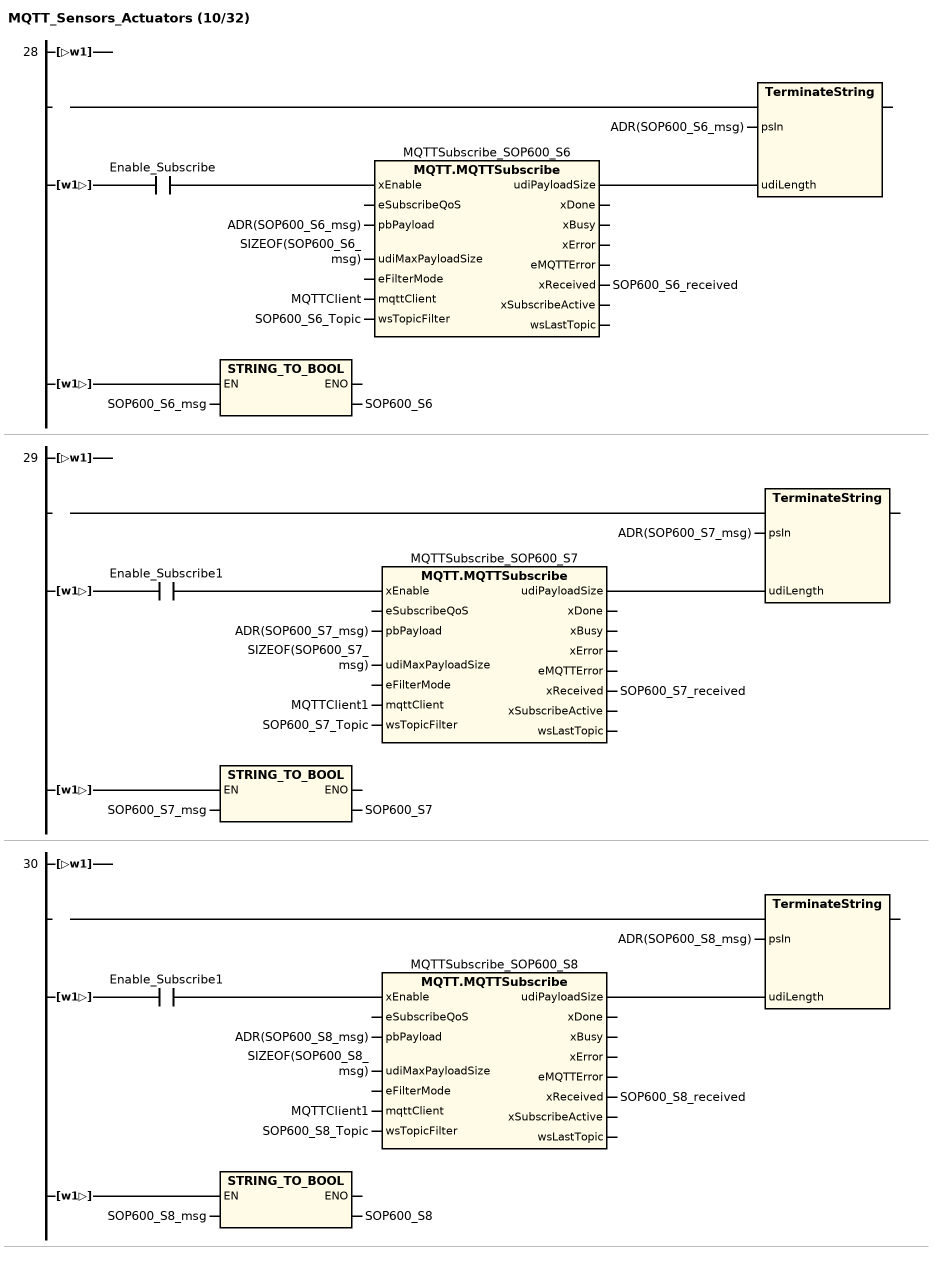
// NETWORK 28
MQTTSubscribe_SOP600_S6(
    xEnable := Enable_Subscribe,
    pbPayload := ADR(SOP600_S6_msg),
    udiMaxPayloadSize := SIZEOF(SOP600_S6_msg),
    mqttClient := MQTTClient,
    wsTopicFilter := SOP600_S6_Topic,
    xReceived => SOP600_S6_received); // MQTT.MQTTSubscribe
TerminateString(psIn := ADR(SOP600_S6_msg), udiLength := MQTTSubscribe_SOP600_S6.udiPayloadSize);
SOP600_S6 := STRING_TO_BOOL(SOP600_S6_msg);

// NETWORK 29
MQTTSubscribe_SOP600_S7(
    xEnable := Enable_Subscribe1,
    pbPayload := ADR(SOP600_S7_msg),
    udiMaxPayloadSize := SIZEOF(SOP600_S7_msg),
    mqttClient := MQTTClient1,
    wsTopicFilter := SOP600_S7_Topic,
    xReceived => SOP600_S7_received); // MQTT.MQTTSubscribe
TerminateString(psIn := ADR(SOP600_S7_msg), udiLength := MQTTSubscribe_SOP600_S7.udiPayloadSize);
SOP600_S7 := STRING_TO_BOOL(SOP600_S7_msg);

// NETWORK 30
MQTTSubscribe_SOP600_S8(
    xEnable := Enable_Subscribe1,
    pbPayload := ADR(SOP600_S8_msg),
    udiMaxPayloadSize := SIZEOF(SOP600_S8_msg),
    mqttClient := MQTTClient1,
    wsTopicFilter := SOP600_S8_Topic,
    xReceived => SOP600_S8_received); // MQTT.MQTTSubscribe
TerminateString(psIn := ADR(SOP600_S8_msg), udiLength := MQTTSubscribe_SOP600_S8.udiPayloadSize);
SOP600_S8 := STRING_TO_BOOL(SOP600_S8_msg);

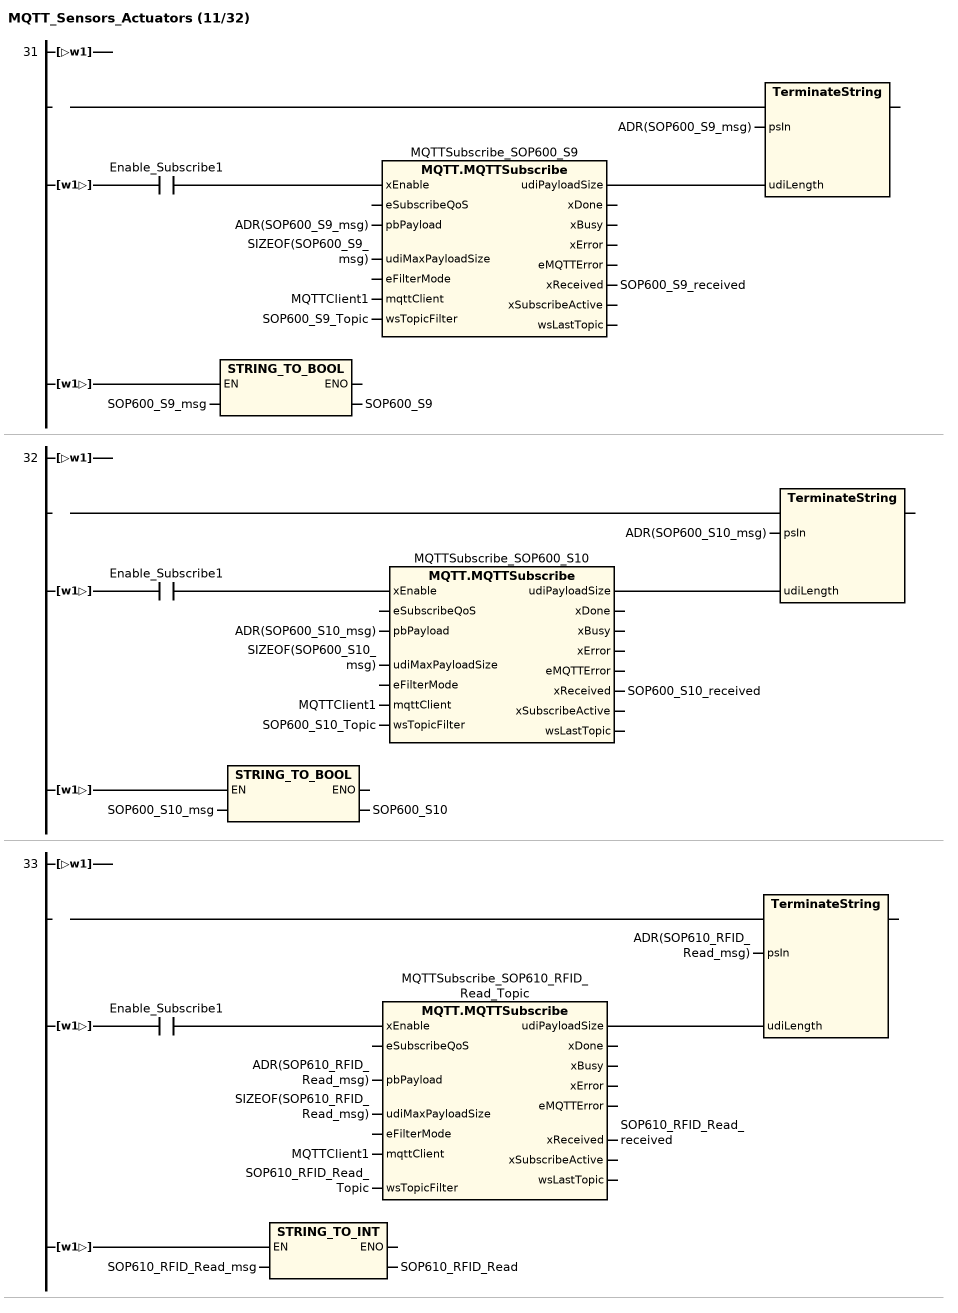
// NETWORK 31
MQTTSubscribe_SOP600_S9(
    xEnable := Enable_Subscribe1,
    pbPayload := ADR(SOP600_S9_msg),
    udiMaxPayloadSize := SIZEOF(SOP600_S9_msg),
    mqttClient := MQTTClient1,
    wsTopicFilter := SOP600_S9_Topic,
    xReceived => SOP600_S9_received); // MQTT.MQTTSubscribe
TerminateString(psIn := ADR(SOP600_S9_msg), udiLength := MQTTSubscribe_SOP600_S9.udiPayloadSize);
SOP600_S9 := STRING_TO_BOOL(SOP600_S9_msg);

// NETWORK 32
MQTTSubscribe_SOP600_S10(
    xEnable := Enable_Subscribe1,
    pbPayload := ADR(SOP600_S10_msg),
    udiMaxPayloadSize := SIZEOF(SOP600_S10_msg),
    mqttClient := MQTTClient1,
    wsTopicFilter := SOP600_S10_Topic,
    xReceived => SOP600_S10_received); // MQTT.MQTTSubscribe
TerminateString(psIn := ADR(SOP600_S10_msg), udiLength := MQTTSubscribe_SOP600_S10.udiPayloadSize);
SOP600_S10 := STRING_TO_BOOL(SOP600_S10_msg);

// NETWORK 33
MQTTSubscribe_SOP610_RFID_Read_Topic(
    xEnable := Enable_Subscribe1,
    pbPayload := ADR(SOP610_RFID_Read_msg),
    udiMaxPayloadSize := SIZEOF(SOP610_RFID_Read_msg),
    mqttClient := MQTTClient1,
    wsTopicFilter := SOP610_RFID_Read_Topic,
    xReceived => SOP610_RFID_Read_received); // MQTT.MQTTSubscribe
TerminateString(psIn := ADR(SOP610_RFID_Read_msg), udiLength := MQTTSubscribe_SOP610_RFID_Read_Topic.udiPayloadSize);
SOP610_RFID_Read := STRING_TO_INT(SOP610_RFID_Read_msg);

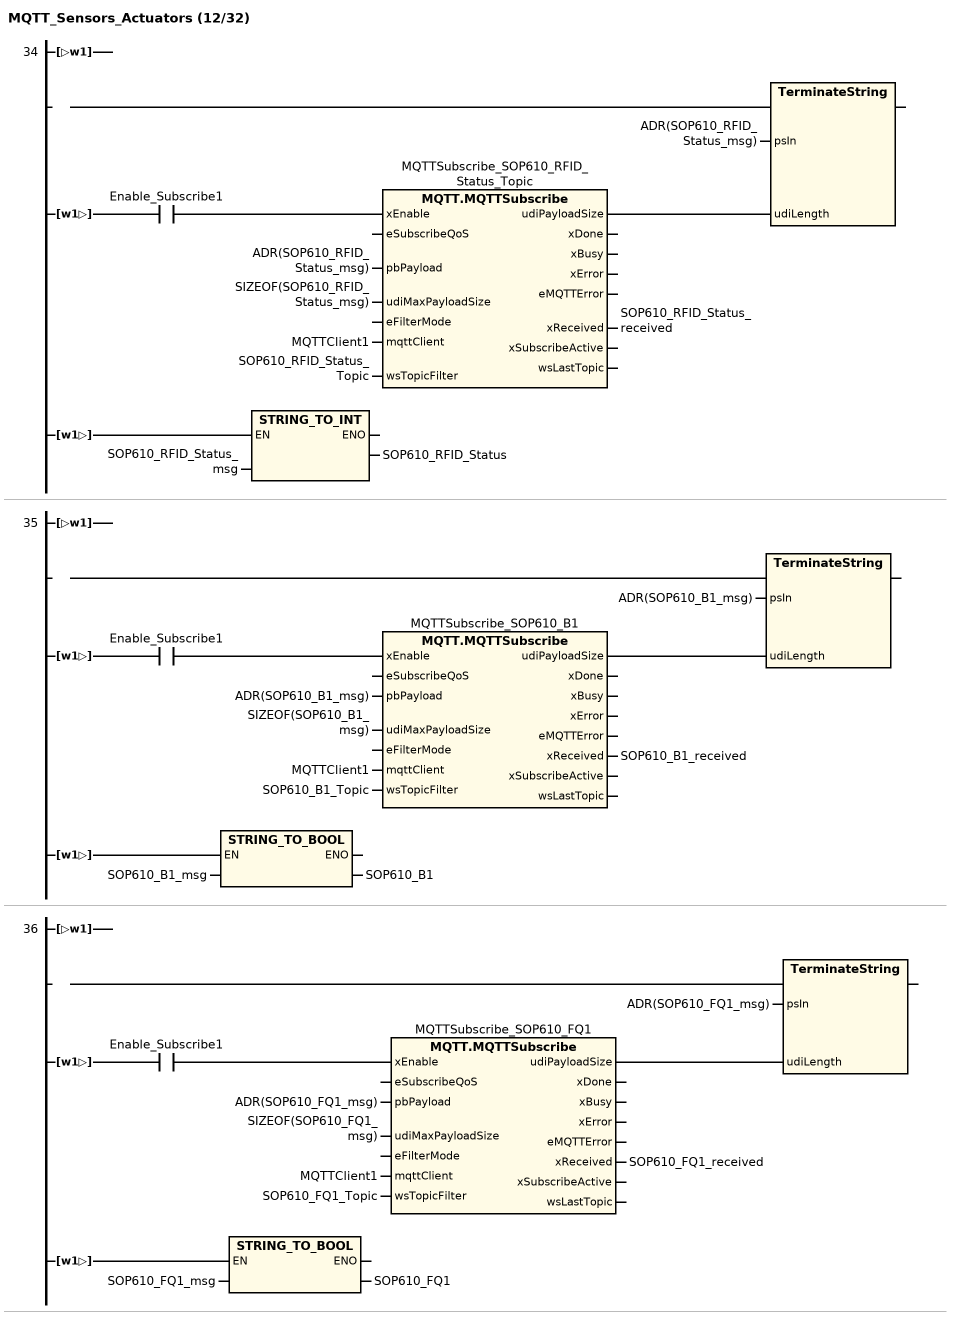
// NETWORK 34
MQTTSubscribe_SOP610_RFID_Status_Topic(
    xEnable := Enable_Subscribe1,
    pbPayload := ADR(SOP610_RFID_Status_msg),
    udiMaxPayloadSize := SIZEOF(SOP610_RFID_Status_msg),
    mqttClient := MQTTClient1,
    wsTopicFilter := SOP610_RFID_Status_Topic,
    xReceived => SOP610_RFID_Status_received); // MQTT.MQTTSubscribe
TerminateString(psIn := ADR(SOP610_RFID_Status_msg), udiLength := MQTTSubscribe_SOP610_RFID_Status_Topic.udiPayloadSize);
SOP610_RFID_Status := STRING_TO_INT(SOP610_RFID_Status_msg);

// NETWORK 35
MQTTSubscribe_SOP610_B1(
    xEnable := Enable_Subscribe1,
    pbPayload := ADR(SOP610_B1_msg),
    udiMaxPayloadSize := SIZEOF(SOP610_B1_msg),
    mqttClient := MQTTClient1,
    wsTopicFilter := SOP610_B1_Topic,
    xReceived => SOP610_B1_received); // MQTT.MQTTSubscribe
TerminateString(psIn := ADR(SOP610_B1_msg), udiLength := MQTTSubscribe_SOP610_B1.udiPayloadSize);
SOP610_B1 := STRING_TO_BOOL(SOP610_B1_msg);

// NETWORK 36
MQTTSubscribe_SOP610_FQ1(
    xEnable := Enable_Subscribe1,
    pbPayload := ADR(SOP610_FQ1_msg),
    udiMaxPayloadSize := SIZEOF(SOP610_FQ1_msg),
    mqttClient := MQTTClient1,
    wsTopicFilter := SOP610_FQ1_Topic,
    xReceived => SOP610_FQ1_received); // MQTT.MQTTSubscribe
TerminateString(psIn := ADR(SOP610_FQ1_msg), udiLength := MQTTSubscribe_SOP610_FQ1.udiPayloadSize);
SOP610_FQ1 := STRING_TO_BOOL(SOP610_FQ1_msg);

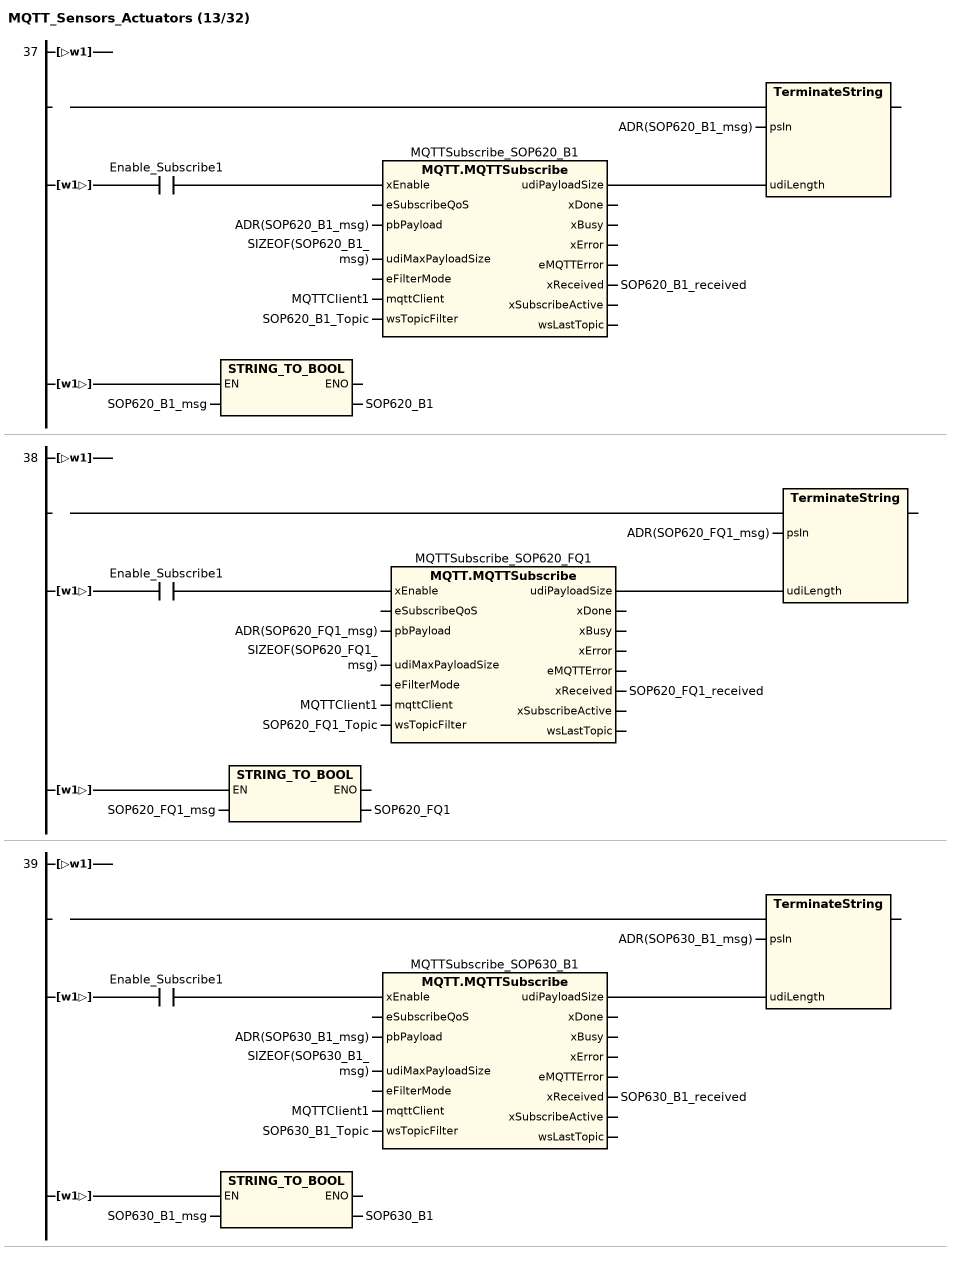
// NETWORK 37
MQTTSubscribe_SOP620_B1(
    xEnable := Enable_Subscribe1,
    pbPayload := ADR(SOP620_B1_msg),
    udiMaxPayloadSize := SIZEOF(SOP620_B1_msg),
    mqttClient := MQTTClient1,
    wsTopicFilter := SOP620_B1_Topic,
    xReceived => SOP620_B1_received); // MQTT.MQTTSubscribe
TerminateString(psIn := ADR(SOP620_B1_msg), udiLength := MQTTSubscribe_SOP620_B1.udiPayloadSize);
SOP620_B1 := STRING_TO_BOOL(SOP620_B1_msg);

// NETWORK 38
MQTTSubscribe_SOP620_FQ1(
    xEnable := Enable_Subscribe1,
    pbPayload := ADR(SOP620_FQ1_msg),
    udiMaxPayloadSize := SIZEOF(SOP620_FQ1_msg),
    mqttClient := MQTTClient1,
    wsTopicFilter := SOP620_FQ1_Topic,
    xReceived => SOP620_FQ1_received); // MQTT.MQTTSubscribe
TerminateString(psIn := ADR(SOP620_FQ1_msg), udiLength := MQTTSubscribe_SOP620_FQ1.udiPayloadSize);
SOP620_FQ1 := STRING_TO_BOOL(SOP620_FQ1_msg);

// NETWORK 39
MQTTSubscribe_SOP630_B1(
    xEnable := Enable_Subscribe1,
    pbPayload := ADR(SOP630_B1_msg),
    udiMaxPayloadSize := SIZEOF(SOP630_B1_msg),
    mqttClient := MQTTClient1,
    wsTopicFilter := SOP630_B1_Topic,
    xReceived => SOP630_B1_received); // MQTT.MQTTSubscribe
TerminateString(psIn := ADR(SOP630_B1_msg), udiLength := MQTTSubscribe_SOP630_B1.udiPayloadSize);
SOP630_B1 := STRING_TO_BOOL(SOP630_B1_msg);

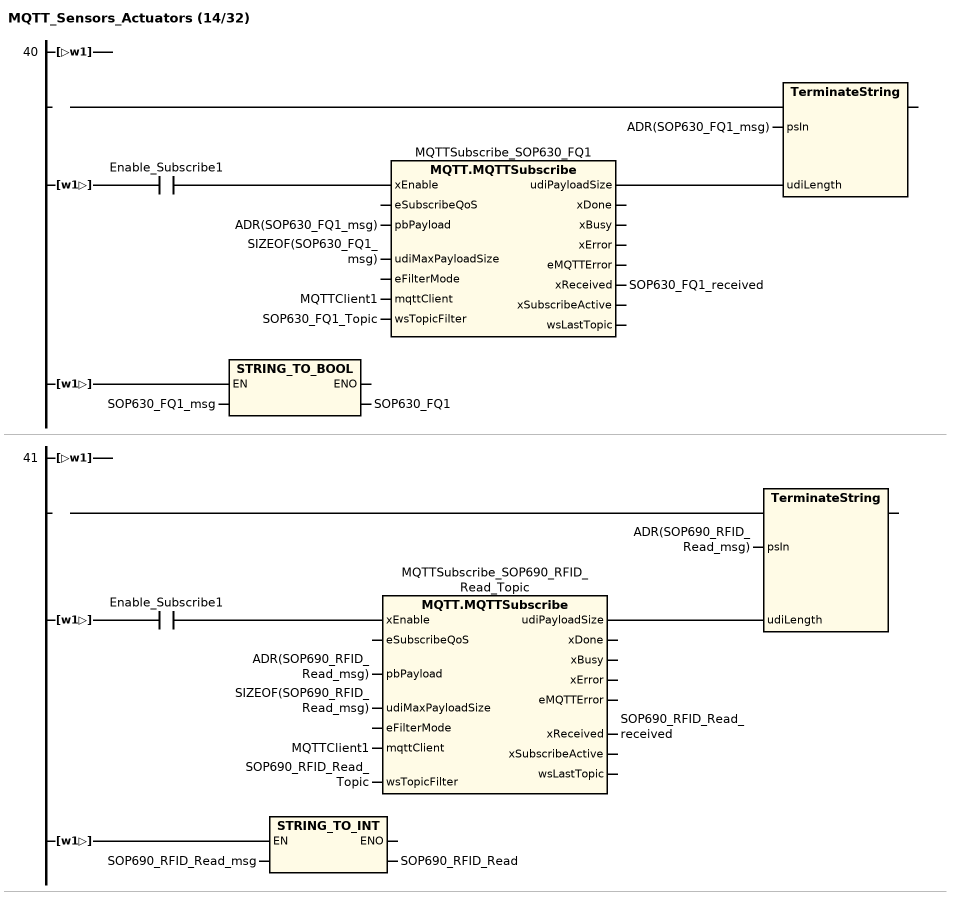
// NETWORK 40
MQTTSubscribe_SOP630_FQ1(
    xEnable := Enable_Subscribe1,
    pbPayload := ADR(SOP630_FQ1_msg),
    udiMaxPayloadSize := SIZEOF(SOP630_FQ1_msg),
    mqttClient := MQTTClient1,
    wsTopicFilter := SOP630_FQ1_Topic,
    xReceived => SOP630_FQ1_received); // MQTT.MQTTSubscribe
TerminateString(psIn := ADR(SOP630_FQ1_msg), udiLength := MQTTSubscribe_SOP630_FQ1.udiPayloadSize);
SOP630_FQ1 := STRING_TO_BOOL(SOP630_FQ1_msg);

// NETWORK 41
MQTTSubscribe_SOP690_RFID_Read_Topic(
    xEnable := Enable_Subscribe1,
    pbPayload := ADR(SOP690_RFID_Read_msg),
    udiMaxPayloadSize := SIZEOF(SOP690_RFID_Read_msg),
    mqttClient := MQTTClient1,
    wsTopicFilter := SOP690_RFID_Read_Topic,
    xReceived => SOP690_RFID_Read_received); // MQTT.MQTTSubscribe
TerminateString(psIn := ADR(SOP690_RFID_Read_msg), udiLength := MQTTSubscribe_SOP690_RFID_Read_Topic.udiPayloadSize);
SOP690_RFID_Read := STRING_TO_INT(SOP690_RFID_Read_msg);

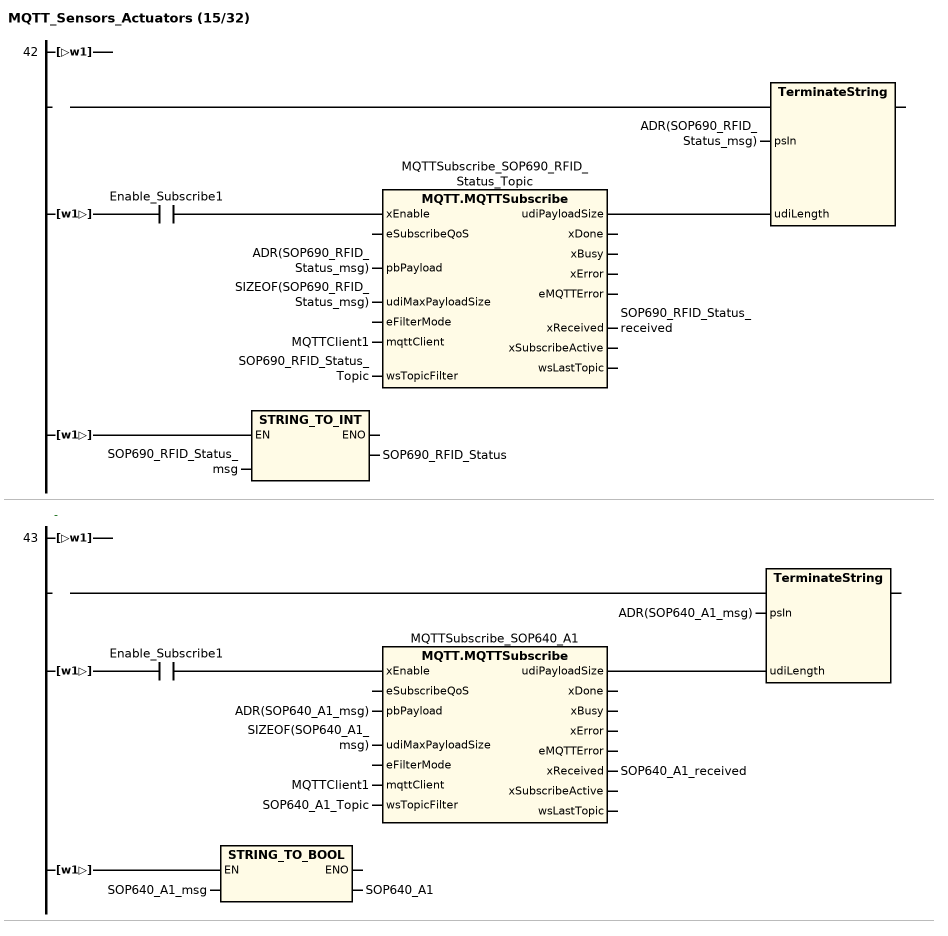
// NETWORK 42
MQTTSubscribe_SOP690_RFID_Status_Topic(
    xEnable := Enable_Subscribe1,
    pbPayload := ADR(SOP690_RFID_Status_msg),
    udiMaxPayloadSize := SIZEOF(SOP690_RFID_Status_msg),
    mqttClient := MQTTClient1,
    wsTopicFilter := SOP690_RFID_Status_Topic,
    xReceived => SOP690_RFID_Status_received); // MQTT.MQTTSubscribe
TerminateString(psIn := ADR(SOP690_RFID_Status_msg), udiLength := MQTTSubscribe_SOP690_RFID_Status_Topic.udiPayloadSize);
SOP690_RFID_Status := STRING_TO_INT(SOP690_RFID_Status_msg);

// NETWORK 43
// -
MQTTSubscribe_SOP640_A1(
    xEnable := Enable_Subscribe1,
    pbPayload := ADR(SOP640_A1_msg),
    udiMaxPayloadSize := SIZEOF(SOP640_A1_msg),
    mqttClient := MQTTClient1,
    wsTopicFilter := SOP640_A1_Topic,
    xReceived => SOP640_A1_received); // MQTT.MQTTSubscribe
TerminateString(psIn := ADR(SOP640_A1_msg), udiLength := MQTTSubscribe_SOP640_A1.udiPayloadSize);
SOP640_A1 := STRING_TO_BOOL(SOP640_A1_msg);

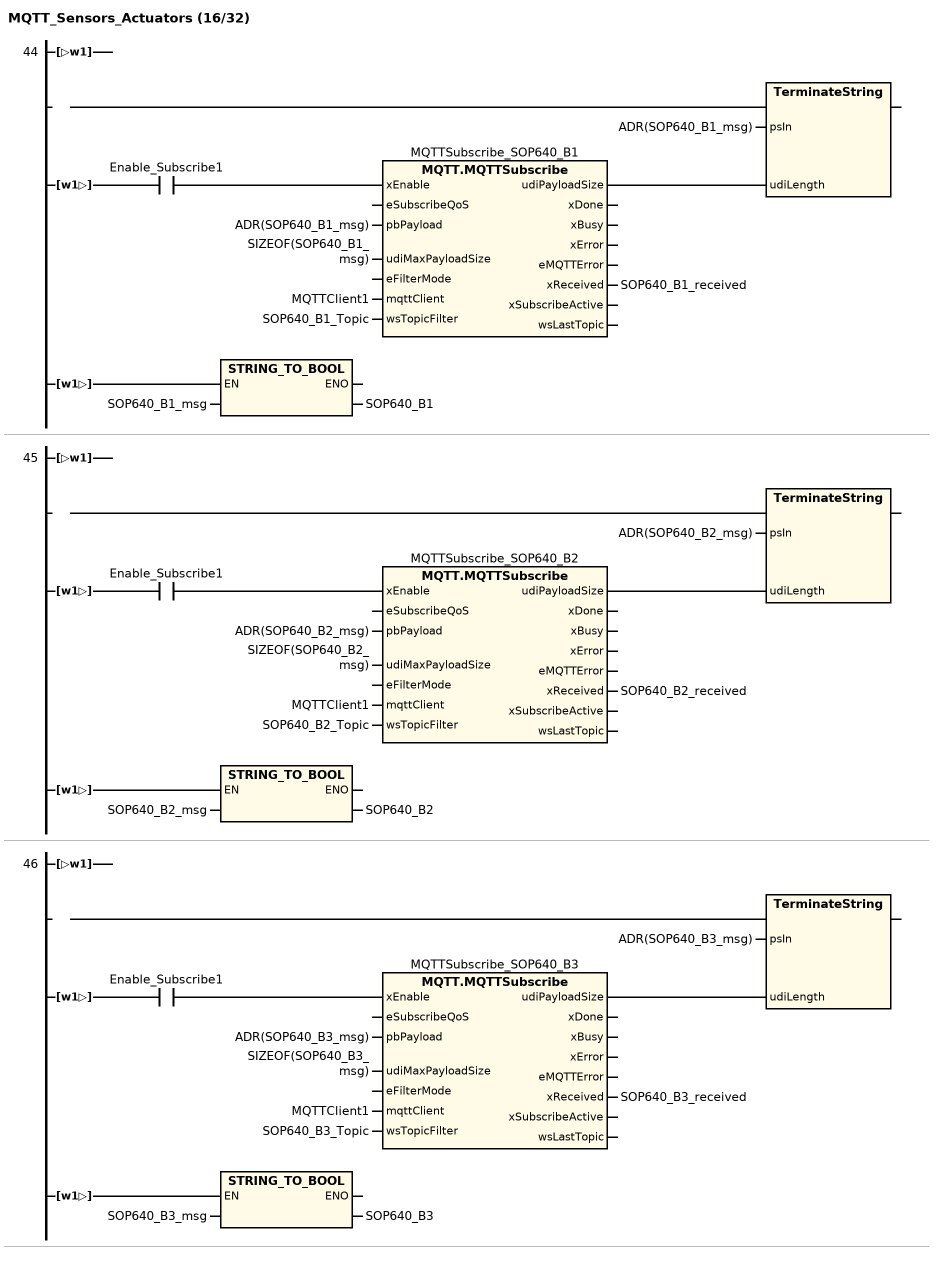
// NETWORK 44
MQTTSubscribe_SOP640_B1(
    xEnable := Enable_Subscribe1,
    pbPayload := ADR(SOP640_B1_msg),
    udiMaxPayloadSize := SIZEOF(SOP640_B1_msg),
    mqttClient := MQTTClient1,
    wsTopicFilter := SOP640_B1_Topic,
    xReceived => SOP640_B1_received); // MQTT.MQTTSubscribe
TerminateString(psIn := ADR(SOP640_B1_msg), udiLength := MQTTSubscribe_SOP640_B1.udiPayloadSize);
SOP640_B1 := STRING_TO_BOOL(SOP640_B1_msg);

// NETWORK 45
MQTTSubscribe_SOP640_B2(
    xEnable := Enable_Subscribe1,
    pbPayload := ADR(SOP640_B2_msg),
    udiMaxPayloadSize := SIZEOF(SOP640_B2_msg),
    mqttClient := MQTTClient1,
    wsTopicFilter := SOP640_B2_Topic,
    xReceived => SOP640_B2_received); // MQTT.MQTTSubscribe
TerminateString(psIn := ADR(SOP640_B2_msg), udiLength := MQTTSubscribe_SOP640_B2.udiPayloadSize);
SOP640_B2 := STRING_TO_BOOL(SOP640_B2_msg);

// NETWORK 46
MQTTSubscribe_SOP640_B3(
    xEnable := Enable_Subscribe1,
    pbPayload := ADR(SOP640_B3_msg),
    udiMaxPayloadSize := SIZEOF(SOP640_B3_msg),
    mqttClient := MQTTClient1,
    wsTopicFilter := SOP640_B3_Topic,
    xReceived => SOP640_B3_received); // MQTT.MQTTSubscribe
TerminateString(psIn := ADR(SOP640_B3_msg), udiLength := MQTTSubscribe_SOP640_B3.udiPayloadSize);
SOP640_B3 := STRING_TO_BOOL(SOP640_B3_msg);

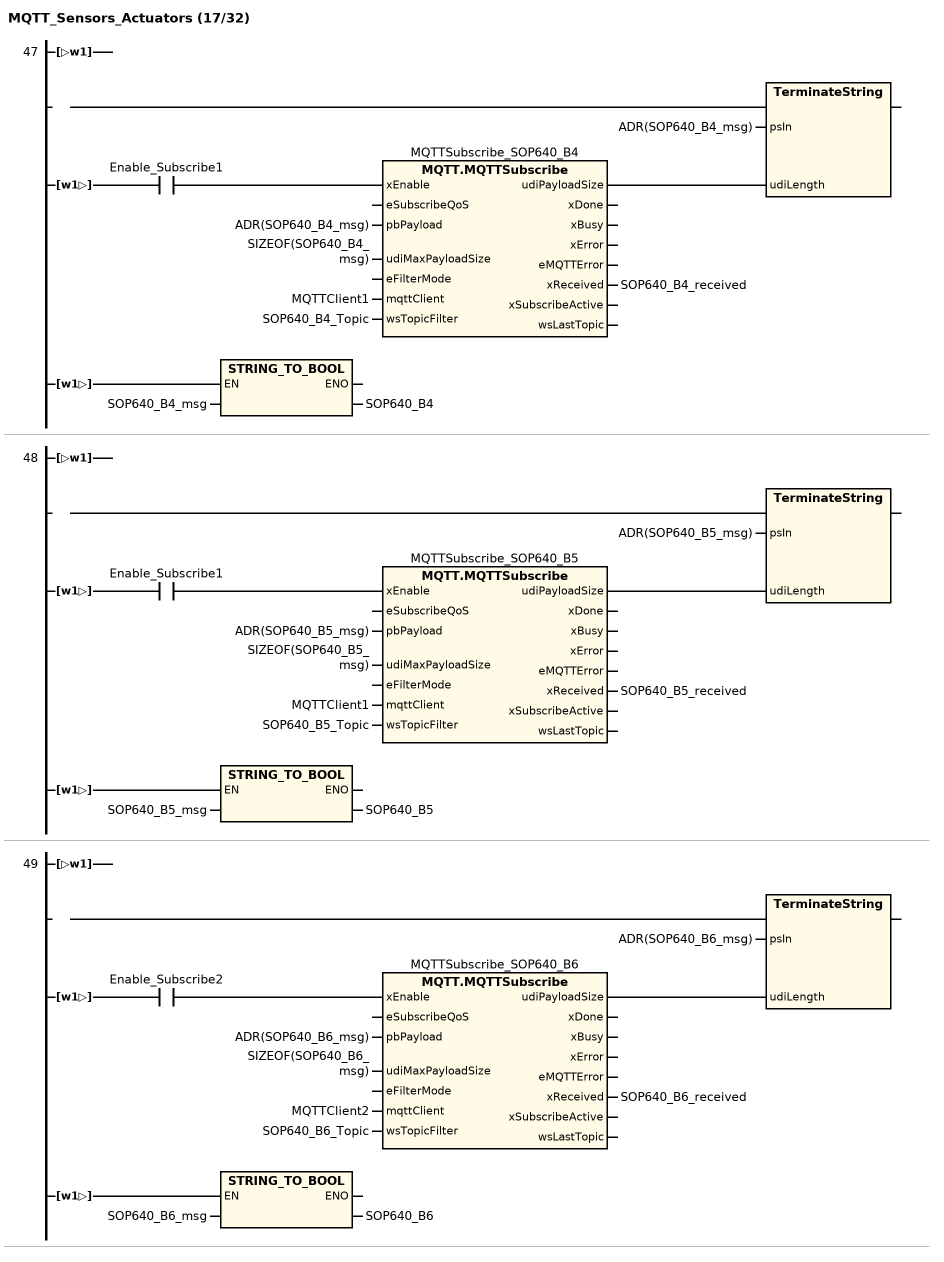
// NETWORK 47
MQTTSubscribe_SOP640_B4(
    xEnable := Enable_Subscribe1,
    pbPayload := ADR(SOP640_B4_msg),
    udiMaxPayloadSize := SIZEOF(SOP640_B4_msg),
    mqttClient := MQTTClient1,
    wsTopicFilter := SOP640_B4_Topic,
    xReceived => SOP640_B4_received); // MQTT.MQTTSubscribe
TerminateString(psIn := ADR(SOP640_B4_msg), udiLength := MQTTSubscribe_SOP640_B4.udiPayloadSize);
SOP640_B4 := STRING_TO_BOOL(SOP640_B4_msg);

// NETWORK 48
MQTTSubscribe_SOP640_B5(
    xEnable := Enable_Subscribe1,
    pbPayload := ADR(SOP640_B5_msg),
    udiMaxPayloadSize := SIZEOF(SOP640_B5_msg),
    mqttClient := MQTTClient1,
    wsTopicFilter := SOP640_B5_Topic,
    xReceived => SOP640_B5_received); // MQTT.MQTTSubscribe
TerminateString(psIn := ADR(SOP640_B5_msg), udiLength := MQTTSubscribe_SOP640_B5.udiPayloadSize);
SOP640_B5 := STRING_TO_BOOL(SOP640_B5_msg);

// NETWORK 49
MQTTSubscribe_SOP640_B6(
    xEnable := Enable_Subscribe2,
    pbPayload := ADR(SOP640_B6_msg),
    udiMaxPayloadSize := SIZEOF(SOP640_B6_msg),
    mqttClient := MQTTClient2,
    wsTopicFilter := SOP640_B6_Topic,
    xReceived => SOP640_B6_received); // MQTT.MQTTSubscribe
TerminateString(psIn := ADR(SOP640_B6_msg), udiLength := MQTTSubscribe_SOP640_B6.udiPayloadSize);
SOP640_B6 := STRING_TO_BOOL(SOP640_B6_msg);

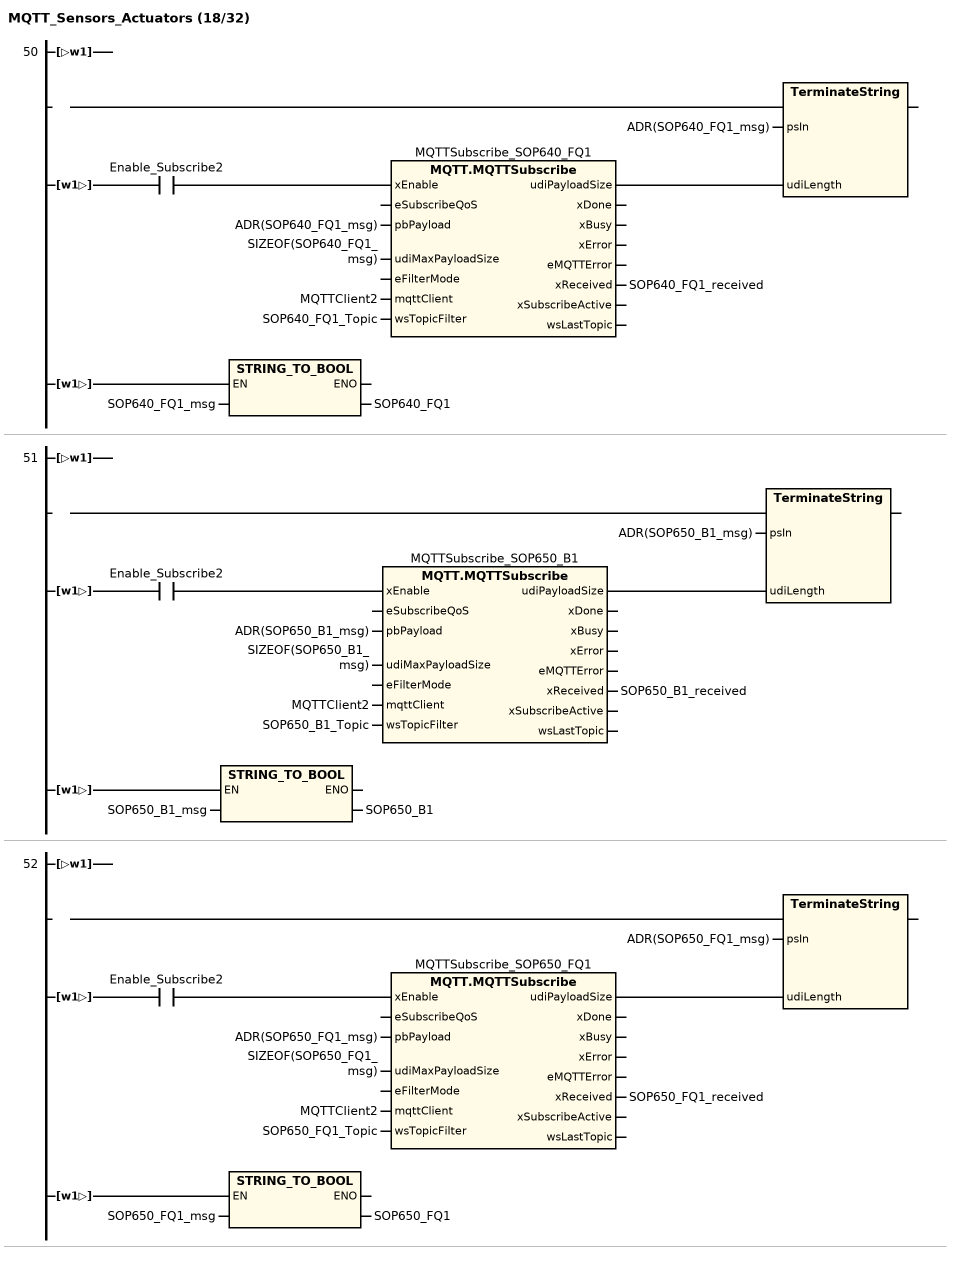
// NETWORK 50
MQTTSubscribe_SOP640_FQ1(
    xEnable := Enable_Subscribe2,
    pbPayload := ADR(SOP640_FQ1_msg),
    udiMaxPayloadSize := SIZEOF(SOP640_FQ1_msg),
    mqttClient := MQTTClient2,
    wsTopicFilter := SOP640_FQ1_Topic,
    xReceived => SOP640_FQ1_received); // MQTT.MQTTSubscribe
TerminateString(psIn := ADR(SOP640_FQ1_msg), udiLength := MQTTSubscribe_SOP640_FQ1.udiPayloadSize);
SOP640_FQ1 := STRING_TO_BOOL(SOP640_FQ1_msg);

// NETWORK 51
MQTTSubscribe_SOP650_B1(
    xEnable := Enable_Subscribe2,
    pbPayload := ADR(SOP650_B1_msg),
    udiMaxPayloadSize := SIZEOF(SOP650_B1_msg),
    mqttClient := MQTTClient2,
    wsTopicFilter := SOP650_B1_Topic,
    xReceived => SOP650_B1_received); // MQTT.MQTTSubscribe
TerminateString(psIn := ADR(SOP650_B1_msg), udiLength := MQTTSubscribe_SOP650_B1.udiPayloadSize);
SOP650_B1 := STRING_TO_BOOL(SOP650_B1_msg);

// NETWORK 52
MQTTSubscribe_SOP650_FQ1(
    xEnable := Enable_Subscribe2,
    pbPayload := ADR(SOP650_FQ1_msg),
    udiMaxPayloadSize := SIZEOF(SOP650_FQ1_msg),
    mqttClient := MQTTClient2,
    wsTopicFilter := SOP650_FQ1_Topic,
    xReceived => SOP650_FQ1_received); // MQTT.MQTTSubscribe
TerminateString(psIn := ADR(SOP650_FQ1_msg), udiLength := MQTTSubscribe_SOP650_FQ1.udiPayloadSize);
SOP650_FQ1 := STRING_TO_BOOL(SOP650_FQ1_msg);

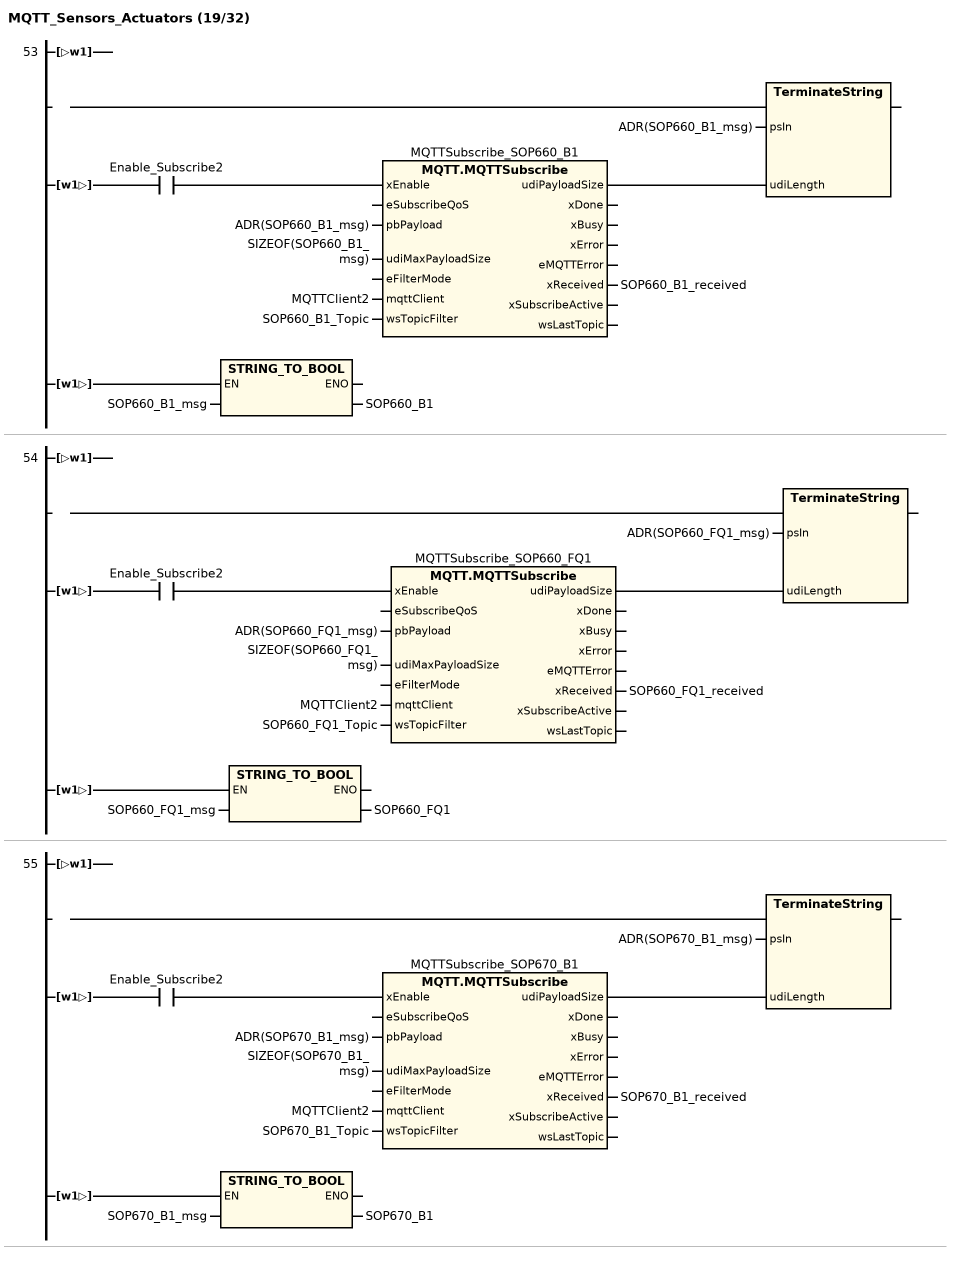
// NETWORK 53
MQTTSubscribe_SOP660_B1(
    xEnable := Enable_Subscribe2,
    pbPayload := ADR(SOP660_B1_msg),
    udiMaxPayloadSize := SIZEOF(SOP660_B1_msg),
    mqttClient := MQTTClient2,
    wsTopicFilter := SOP660_B1_Topic,
    xReceived => SOP660_B1_received); // MQTT.MQTTSubscribe
TerminateString(psIn := ADR(SOP660_B1_msg), udiLength := MQTTSubscribe_SOP660_B1.udiPayloadSize);
SOP660_B1 := STRING_TO_BOOL(SOP660_B1_msg);

// NETWORK 54
MQTTSubscribe_SOP660_FQ1(
    xEnable := Enable_Subscribe2,
    pbPayload := ADR(SOP660_FQ1_msg),
    udiMaxPayloadSize := SIZEOF(SOP660_FQ1_msg),
    mqttClient := MQTTClient2,
    wsTopicFilter := SOP660_FQ1_Topic,
    xReceived => SOP660_FQ1_received); // MQTT.MQTTSubscribe
TerminateString(psIn := ADR(SOP660_FQ1_msg), udiLength := MQTTSubscribe_SOP660_FQ1.udiPayloadSize);
SOP660_FQ1 := STRING_TO_BOOL(SOP660_FQ1_msg);

// NETWORK 55
MQTTSubscribe_SOP670_B1(
    xEnable := Enable_Subscribe2,
    pbPayload := ADR(SOP670_B1_msg),
    udiMaxPayloadSize := SIZEOF(SOP670_B1_msg),
    mqttClient := MQTTClient2,
    wsTopicFilter := SOP670_B1_Topic,
    xReceived => SOP670_B1_received); // MQTT.MQTTSubscribe
TerminateString(psIn := ADR(SOP670_B1_msg), udiLength := MQTTSubscribe_SOP670_B1.udiPayloadSize);
SOP670_B1 := STRING_TO_BOOL(SOP670_B1_msg);

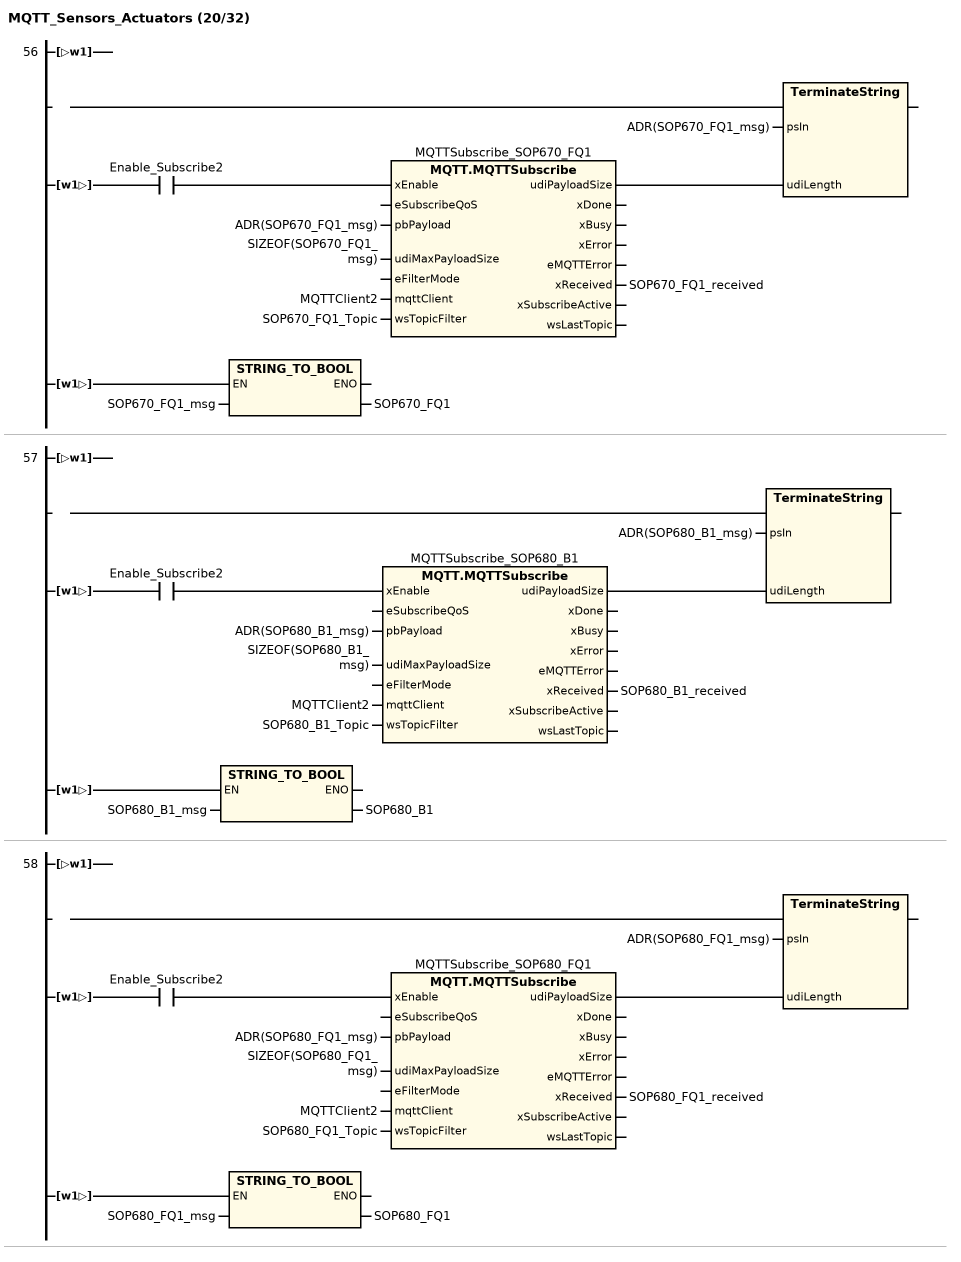
// NETWORK 56
MQTTSubscribe_SOP670_FQ1(
    xEnable := Enable_Subscribe2,
    pbPayload := ADR(SOP670_FQ1_msg),
    udiMaxPayloadSize := SIZEOF(SOP670_FQ1_msg),
    mqttClient := MQTTClient2,
    wsTopicFilter := SOP670_FQ1_Topic,
    xReceived => SOP670_FQ1_received); // MQTT.MQTTSubscribe
TerminateString(psIn := ADR(SOP670_FQ1_msg), udiLength := MQTTSubscribe_SOP670_FQ1.udiPayloadSize);
SOP670_FQ1 := STRING_TO_BOOL(SOP670_FQ1_msg);

// NETWORK 57
MQTTSubscribe_SOP680_B1(
    xEnable := Enable_Subscribe2,
    pbPayload := ADR(SOP680_B1_msg),
    udiMaxPayloadSize := SIZEOF(SOP680_B1_msg),
    mqttClient := MQTTClient2,
    wsTopicFilter := SOP680_B1_Topic,
    xReceived => SOP680_B1_received); // MQTT.MQTTSubscribe
TerminateString(psIn := ADR(SOP680_B1_msg), udiLength := MQTTSubscribe_SOP680_B1.udiPayloadSize);
SOP680_B1 := STRING_TO_BOOL(SOP680_B1_msg);

// NETWORK 58
MQTTSubscribe_SOP680_FQ1(
    xEnable := Enable_Subscribe2,
    pbPayload := ADR(SOP680_FQ1_msg),
    udiMaxPayloadSize := SIZEOF(SOP680_FQ1_msg),
    mqttClient := MQTTClient2,
    wsTopicFilter := SOP680_FQ1_Topic,
    xReceived => SOP680_FQ1_received); // MQTT.MQTTSubscribe
TerminateString(psIn := ADR(SOP680_FQ1_msg), udiLength := MQTTSubscribe_SOP680_FQ1.udiPayloadSize);
SOP680_FQ1 := STRING_TO_BOOL(SOP680_FQ1_msg);

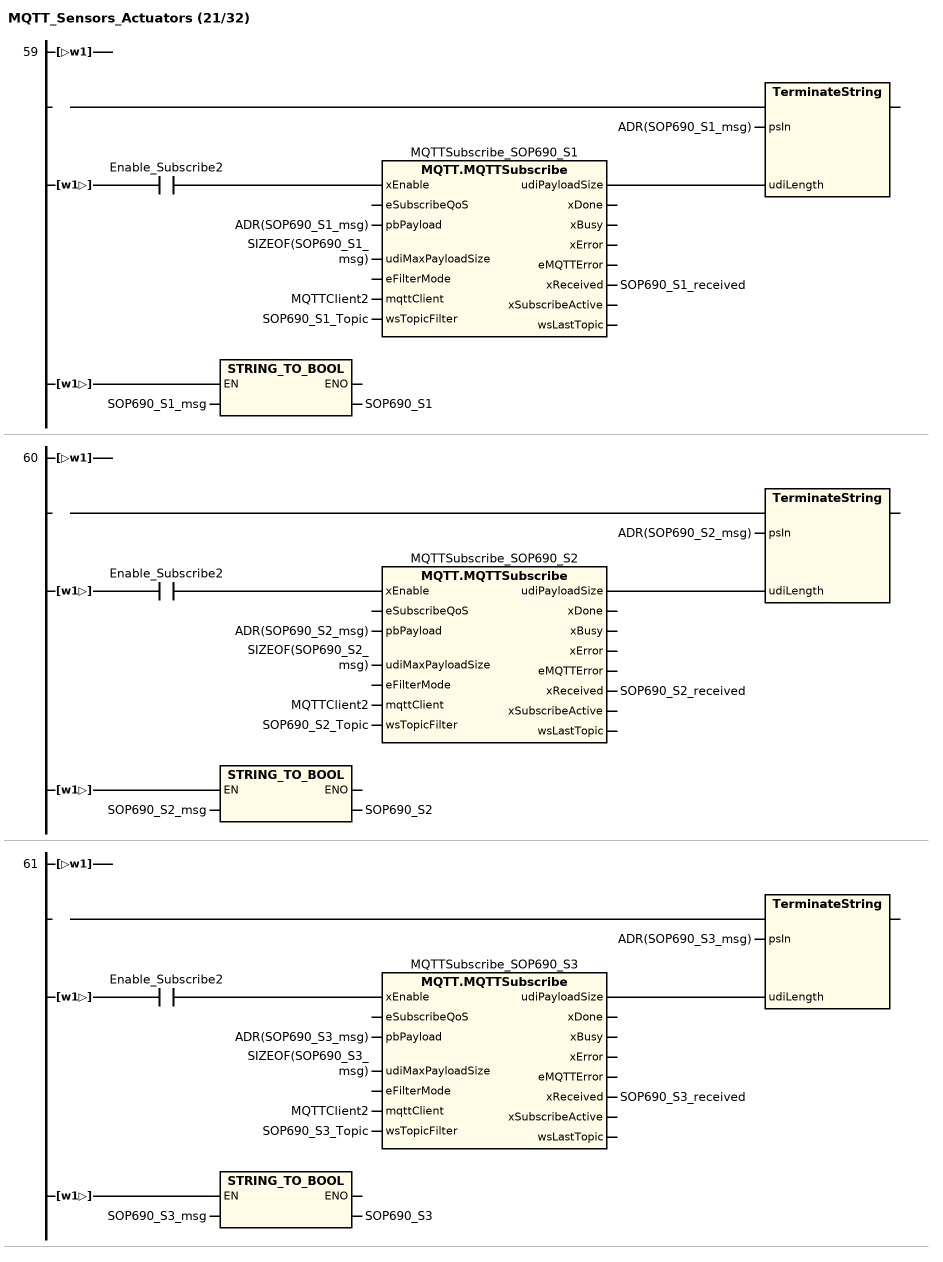
// NETWORK 59
MQTTSubscribe_SOP690_S1(
    xEnable := Enable_Subscribe2,
    pbPayload := ADR(SOP690_S1_msg),
    udiMaxPayloadSize := SIZEOF(SOP690_S1_msg),
    mqttClient := MQTTClient2,
    wsTopicFilter := SOP690_S1_Topic,
    xReceived => SOP690_S1_received); // MQTT.MQTTSubscribe
TerminateString(psIn := ADR(SOP690_S1_msg), udiLength := MQTTSubscribe_SOP690_S1.udiPayloadSize);
SOP690_S1 := STRING_TO_BOOL(SOP690_S1_msg);

// NETWORK 60
MQTTSubscribe_SOP690_S2(
    xEnable := Enable_Subscribe2,
    pbPayload := ADR(SOP690_S2_msg),
    udiMaxPayloadSize := SIZEOF(SOP690_S2_msg),
    mqttClient := MQTTClient2,
    wsTopicFilter := SOP690_S2_Topic,
    xReceived => SOP690_S2_received); // MQTT.MQTTSubscribe
TerminateString(psIn := ADR(SOP690_S2_msg), udiLength := MQTTSubscribe_SOP690_S2.udiPayloadSize);
SOP690_S2 := STRING_TO_BOOL(SOP690_S2_msg);

// NETWORK 61
MQTTSubscribe_SOP690_S3(
    xEnable := Enable_Subscribe2,
    pbPayload := ADR(SOP690_S3_msg),
    udiMaxPayloadSize := SIZEOF(SOP690_S3_msg),
    mqttClient := MQTTClient2,
    wsTopicFilter := SOP690_S3_Topic,
    xReceived => SOP690_S3_received); // MQTT.MQTTSubscribe
TerminateString(psIn := ADR(SOP690_S3_msg), udiLength := MQTTSubscribe_SOP690_S3.udiPayloadSize);
SOP690_S3 := STRING_TO_BOOL(SOP690_S3_msg);

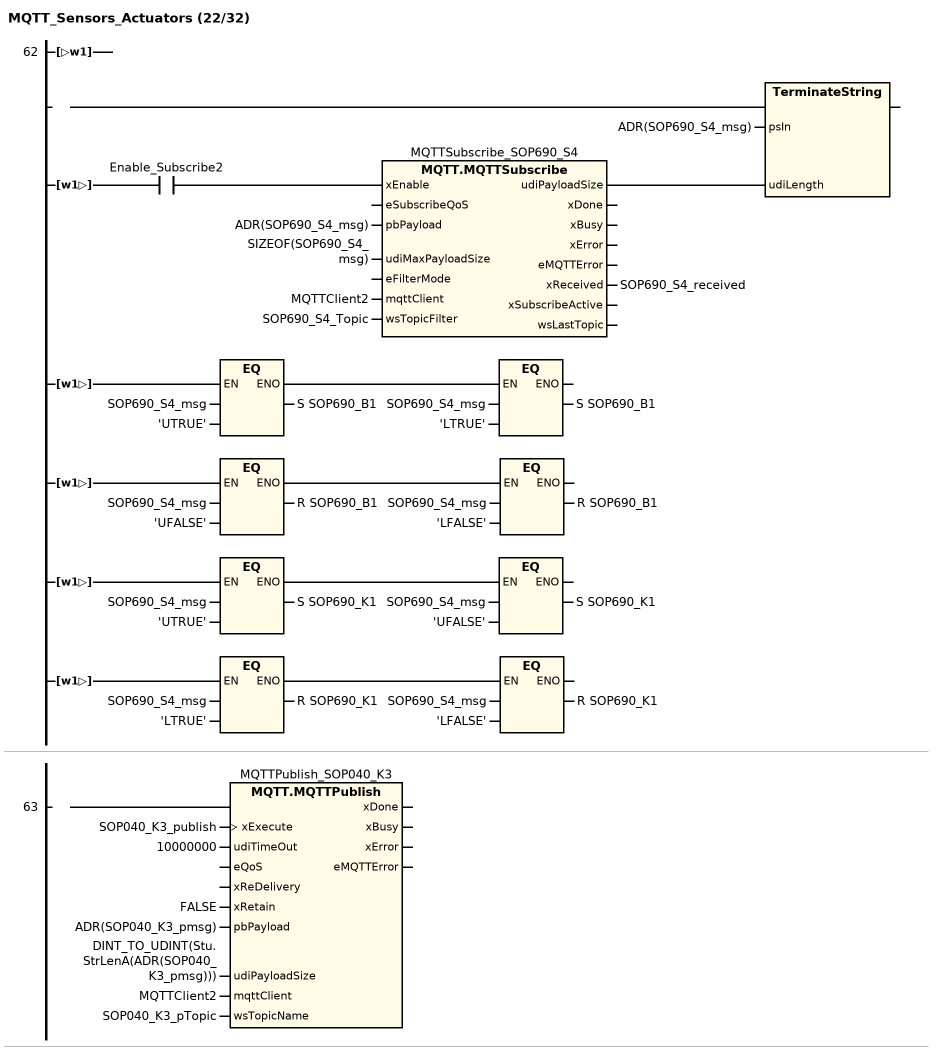
// NETWORK 62
MQTTSubscribe_SOP690_S4(
    xEnable := Enable_Subscribe2,
    pbPayload := ADR(SOP690_S4_msg),
    udiMaxPayloadSize := SIZEOF(SOP690_S4_msg),
    mqttClient := MQTTClient2,
    wsTopicFilter := SOP690_S4_Topic,
    xReceived => SOP690_S4_received); // MQTT.MQTTSubscribe
TerminateString(psIn := ADR(SOP690_S4_msg), udiLength := MQTTSubscribe_SOP690_S4.udiPayloadSize);
SOP690_B1 S= SOP690_S4_msg = 'UTRUE';
SOP690_B1 S= SOP690_S4_msg = 'LTRUE';
SOP690_B1 R= SOP690_S4_msg = 'UFALSE';
SOP690_B1 R= SOP690_S4_msg = 'LFALSE';
SOP690_K1 S= SOP690_S4_msg = 'UTRUE';
SOP690_K1 S= SOP690_S4_msg = 'UFALSE';
SOP690_K1 R= SOP690_S4_msg = 'LTRUE';
SOP690_K1 R= SOP690_S4_msg = 'LFALSE';

// NETWORK 63
_rt13(CLK := SOP040_K3_publish);
MQTTPublish_SOP040_K3(
    xExecute := _rt13.Q,
    udiTimeOut := 10000000,
    xRetain := FALSE,
    pbPayload := ADR(SOP040_K3_pmsg),
    udiPayloadSize := DINT_TO_UDINT(Stu.StrLenA(ADR(SOP040_K3_pmsg))),
    mqttClient := MQTTClient2,
    wsTopicName := SOP040_K3_pTopic); // MQTT.MQTTPublish

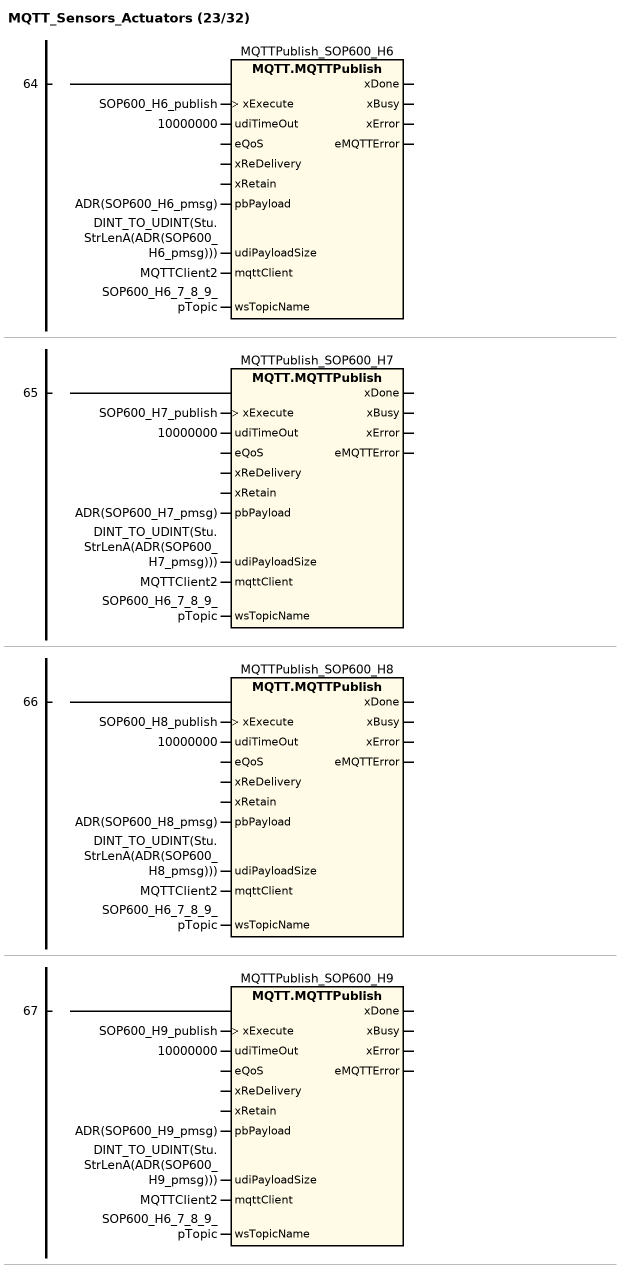
// NETWORK 64
_rt14(CLK := SOP600_H6_publish);
MQTTPublish_SOP600_H6(
    xExecute := _rt14.Q,
    udiTimeOut := 10000000,
    pbPayload := ADR(SOP600_H6_pmsg),
    udiPayloadSize := DINT_TO_UDINT(Stu.StrLenA(ADR(SOP600_H6_pmsg))),
    mqttClient := MQTTClient2,
    wsTopicName := SOP600_H6_7_8_9_pTopic); // MQTT.MQTTPublish

// NETWORK 65
_rt15(CLK := SOP600_H7_publish);
MQTTPublish_SOP600_H7(
    xExecute := _rt15.Q,
    udiTimeOut := 10000000,
    pbPayload := ADR(SOP600_H7_pmsg),
    udiPayloadSize := DINT_TO_UDINT(Stu.StrLenA(ADR(SOP600_H7_pmsg))),
    mqttClient := MQTTClient2,
    wsTopicName := SOP600_H6_7_8_9_pTopic); // MQTT.MQTTPublish

// NETWORK 66
_rt16(CLK := SOP600_H8_publish);
MQTTPublish_SOP600_H8(
    xExecute := _rt16.Q,
    udiTimeOut := 10000000,
    pbPayload := ADR(SOP600_H8_pmsg),
    udiPayloadSize := DINT_TO_UDINT(Stu.StrLenA(ADR(SOP600_H8_pmsg))),
    mqttClient := MQTTClient2,
    wsTopicName := SOP600_H6_7_8_9_pTopic); // MQTT.MQTTPublish

// NETWORK 67
_rt17(CLK := SOP600_H9_publish);
MQTTPublish_SOP600_H9(
    xExecute := _rt17.Q,
    udiTimeOut := 10000000,
    pbPayload := ADR(SOP600_H9_pmsg),
    udiPayloadSize := DINT_TO_UDINT(Stu.StrLenA(ADR(SOP600_H9_pmsg))),
    mqttClient := MQTTClient2,
    wsTopicName := SOP600_H6_7_8_9_pTopic); // MQTT.MQTTPublish

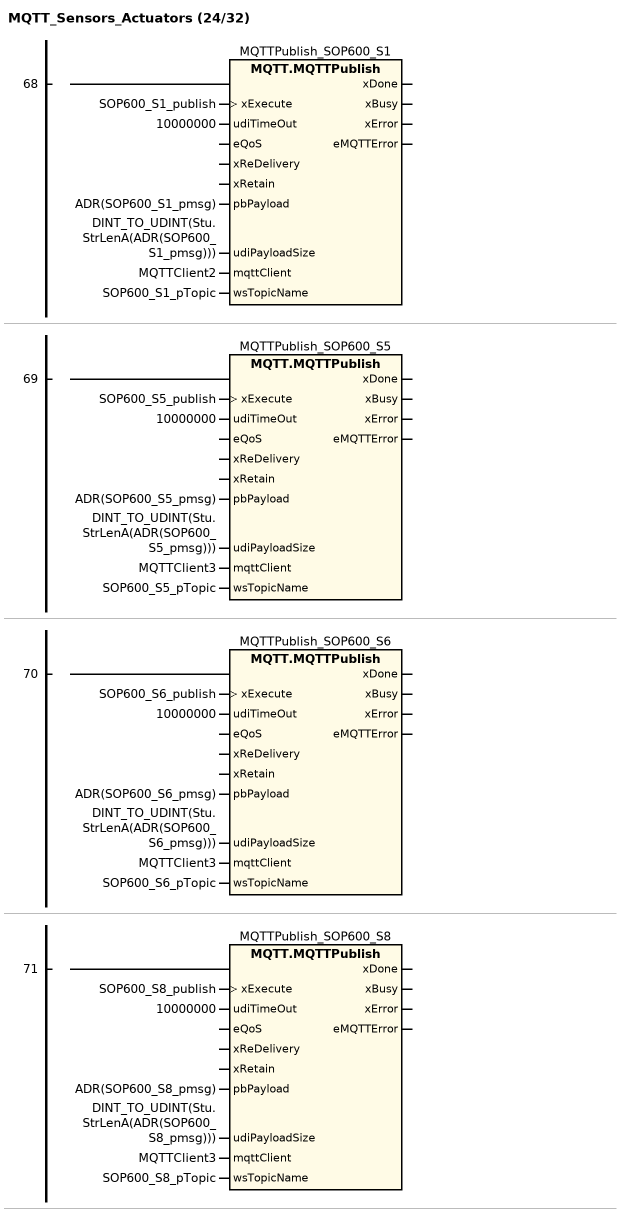
// NETWORK 68
_rt18(CLK := SOP600_S1_publish);
MQTTPublish_SOP600_S1(
    xExecute := _rt18.Q,
    udiTimeOut := 10000000,
    pbPayload := ADR(SOP600_S1_pmsg),
    udiPayloadSize := DINT_TO_UDINT(Stu.StrLenA(ADR(SOP600_S1_pmsg))),
    mqttClient := MQTTClient2,
    wsTopicName := SOP600_S1_pTopic); // MQTT.MQTTPublish

// NETWORK 69
_rt19(CLK := SOP600_S5_publish);
MQTTPublish_SOP600_S5(
    xExecute := _rt19.Q,
    udiTimeOut := 10000000,
    pbPayload := ADR(SOP600_S5_pmsg),
    udiPayloadSize := DINT_TO_UDINT(Stu.StrLenA(ADR(SOP600_S5_pmsg))),
    mqttClient := MQTTClient3,
    wsTopicName := SOP600_S5_pTopic); // MQTT.MQTTPublish

// NETWORK 70
_rt20(CLK := SOP600_S6_publish);
MQTTPublish_SOP600_S6(
    xExecute := _rt20.Q,
    udiTimeOut := 10000000,
    pbPayload := ADR(SOP600_S6_pmsg),
    udiPayloadSize := DINT_TO_UDINT(Stu.StrLenA(ADR(SOP600_S6_pmsg))),
    mqttClient := MQTTClient3,
    wsTopicName := SOP600_S6_pTopic); // MQTT.MQTTPublish

// NETWORK 71
_rt21(CLK := SOP600_S8_publish);
MQTTPublish_SOP600_S8(
    xExecute := _rt21.Q,
    udiTimeOut := 10000000,
    pbPayload := ADR(SOP600_S8_pmsg),
    udiPayloadSize := DINT_TO_UDINT(Stu.StrLenA(ADR(SOP600_S8_pmsg))),
    mqttClient := MQTTClient3,
    wsTopicName := SOP600_S8_pTopic); // MQTT.MQTTPublish

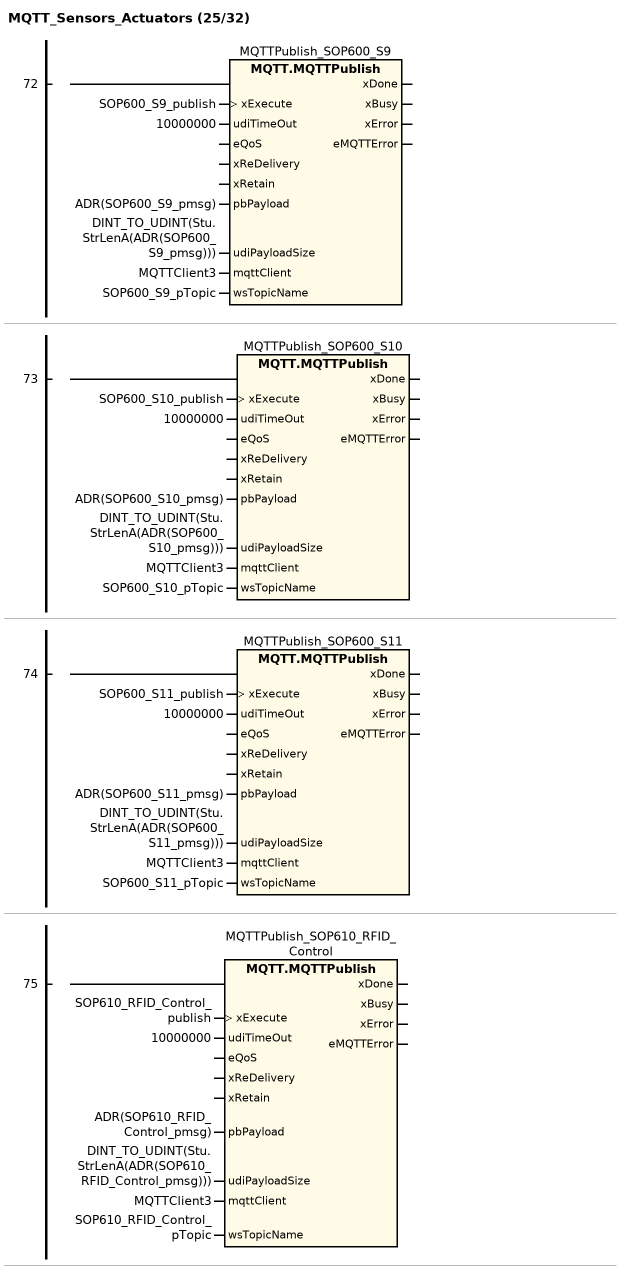
// NETWORK 72
_rt22(CLK := SOP600_S9_publish);
MQTTPublish_SOP600_S9(
    xExecute := _rt22.Q,
    udiTimeOut := 10000000,
    pbPayload := ADR(SOP600_S9_pmsg),
    udiPayloadSize := DINT_TO_UDINT(Stu.StrLenA(ADR(SOP600_S9_pmsg))),
    mqttClient := MQTTClient3,
    wsTopicName := SOP600_S9_pTopic); // MQTT.MQTTPublish

// NETWORK 73
_rt23(CLK := SOP600_S10_publish);
MQTTPublish_SOP600_S10(
    xExecute := _rt23.Q,
    udiTimeOut := 10000000,
    pbPayload := ADR(SOP600_S10_pmsg),
    udiPayloadSize := DINT_TO_UDINT(Stu.StrLenA(ADR(SOP600_S10_pmsg))),
    mqttClient := MQTTClient3,
    wsTopicName := SOP600_S10_pTopic); // MQTT.MQTTPublish

// NETWORK 74
_rt24(CLK := SOP600_S11_publish);
MQTTPublish_SOP600_S11(
    xExecute := _rt24.Q,
    udiTimeOut := 10000000,
    pbPayload := ADR(SOP600_S11_pmsg),
    udiPayloadSize := DINT_TO_UDINT(Stu.StrLenA(ADR(SOP600_S11_pmsg))),
    mqttClient := MQTTClient3,
    wsTopicName := SOP600_S11_pTopic); // MQTT.MQTTPublish

// NETWORK 75
_rt25(CLK := SOP610_RFID_Control_publish);
MQTTPublish_SOP610_RFID_Control(
    xExecute := _rt25.Q,
    udiTimeOut := 10000000,
    pbPayload := ADR(SOP610_RFID_Control_pmsg),
    udiPayloadSize := DINT_TO_UDINT(Stu.StrLenA(ADR(SOP610_RFID_Control_pmsg))),
    mqttClient := MQTTClient3,
    wsTopicName := SOP610_RFID_Control_pTopic); // MQTT.MQTTPublish

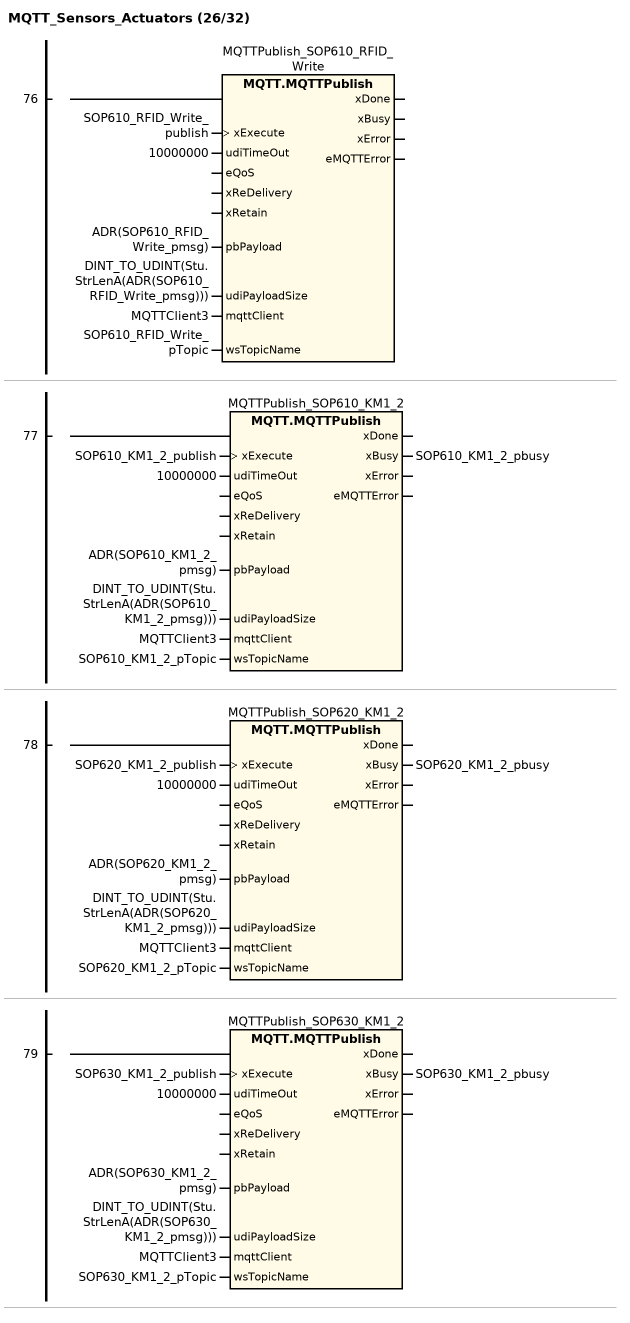
// NETWORK 76
_rt26(CLK := SOP610_RFID_Write_publish);
MQTTPublish_SOP610_RFID_Write(
    xExecute := _rt26.Q,
    udiTimeOut := 10000000,
    pbPayload := ADR(SOP610_RFID_Write_pmsg),
    udiPayloadSize := DINT_TO_UDINT(Stu.StrLenA(ADR(SOP610_RFID_Write_pmsg))),
    mqttClient := MQTTClient3,
    wsTopicName := SOP610_RFID_Write_pTopic); // MQTT.MQTTPublish

// NETWORK 77
_rt27(CLK := SOP610_KM1_2_publish);
MQTTPublish_SOP610_KM1_2(
    xExecute := _rt27.Q,
    udiTimeOut := 10000000,
    pbPayload := ADR(SOP610_KM1_2_pmsg),
    udiPayloadSize := DINT_TO_UDINT(Stu.StrLenA(ADR(SOP610_KM1_2_pmsg))),
    mqttClient := MQTTClient3,
    wsTopicName := SOP610_KM1_2_pTopic,
    xBusy => SOP610_KM1_2_pbusy); // MQTT.MQTTPublish

// NETWORK 78
_rt28(CLK := SOP620_KM1_2_publish);
MQTTPublish_SOP620_KM1_2(
    xExecute := _rt28.Q,
    udiTimeOut := 10000000,
    pbPayload := ADR(SOP620_KM1_2_pmsg),
    udiPayloadSize := DINT_TO_UDINT(Stu.StrLenA(ADR(SOP620_KM1_2_pmsg))),
    mqttClient := MQTTClient3,
    wsTopicName := SOP620_KM1_2_pTopic,
    xBusy => SOP620_KM1_2_pbusy); // MQTT.MQTTPublish

// NETWORK 79
_rt29(CLK := SOP630_KM1_2_publish);
MQTTPublish_SOP630_KM1_2(
    xExecute := _rt29.Q,
    udiTimeOut := 10000000,
    pbPayload := ADR(SOP630_KM1_2_pmsg),
    udiPayloadSize := DINT_TO_UDINT(Stu.StrLenA(ADR(SOP630_KM1_2_pmsg))),
    mqttClient := MQTTClient3,
    wsTopicName := SOP630_KM1_2_pTopic,
    xBusy => SOP630_KM1_2_pbusy); // MQTT.MQTTPublish

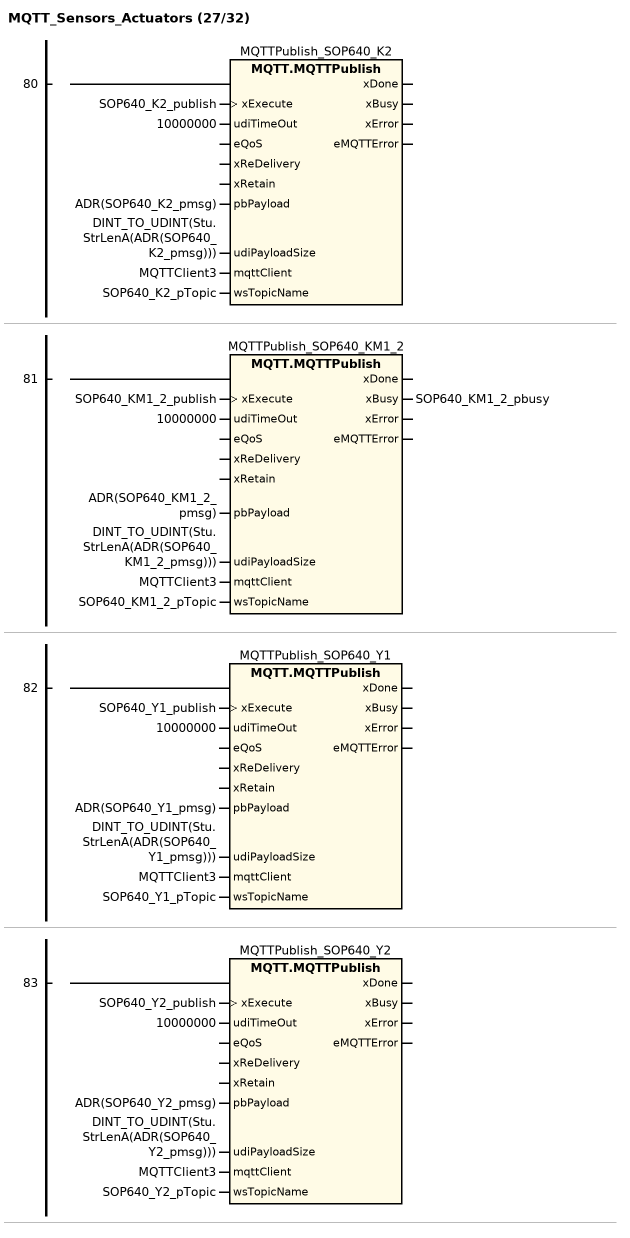
// NETWORK 80
_rt30(CLK := SOP640_K2_publish);
MQTTPublish_SOP640_K2(
    xExecute := _rt30.Q,
    udiTimeOut := 10000000,
    pbPayload := ADR(SOP640_K2_pmsg),
    udiPayloadSize := DINT_TO_UDINT(Stu.StrLenA(ADR(SOP640_K2_pmsg))),
    mqttClient := MQTTClient3,
    wsTopicName := SOP640_K2_pTopic); // MQTT.MQTTPublish

// NETWORK 81
_rt31(CLK := SOP640_KM1_2_publish);
MQTTPublish_SOP640_KM1_2(
    xExecute := _rt31.Q,
    udiTimeOut := 10000000,
    pbPayload := ADR(SOP640_KM1_2_pmsg),
    udiPayloadSize := DINT_TO_UDINT(Stu.StrLenA(ADR(SOP640_KM1_2_pmsg))),
    mqttClient := MQTTClient3,
    wsTopicName := SOP640_KM1_2_pTopic,
    xBusy => SOP640_KM1_2_pbusy); // MQTT.MQTTPublish

// NETWORK 82
_rt32(CLK := SOP640_Y1_publish);
MQTTPublish_SOP640_Y1(
    xExecute := _rt32.Q,
    udiTimeOut := 10000000,
    pbPayload := ADR(SOP640_Y1_pmsg),
    udiPayloadSize := DINT_TO_UDINT(Stu.StrLenA(ADR(SOP640_Y1_pmsg))),
    mqttClient := MQTTClient3,
    wsTopicName := SOP640_Y1_pTopic); // MQTT.MQTTPublish

// NETWORK 83
_rt33(CLK := SOP640_Y2_publish);
MQTTPublish_SOP640_Y2(
    xExecute := _rt33.Q,
    udiTimeOut := 10000000,
    pbPayload := ADR(SOP640_Y2_pmsg),
    udiPayloadSize := DINT_TO_UDINT(Stu.StrLenA(ADR(SOP640_Y2_pmsg))),
    mqttClient := MQTTClient3,
    wsTopicName := SOP640_Y2_pTopic); // MQTT.MQTTPublish

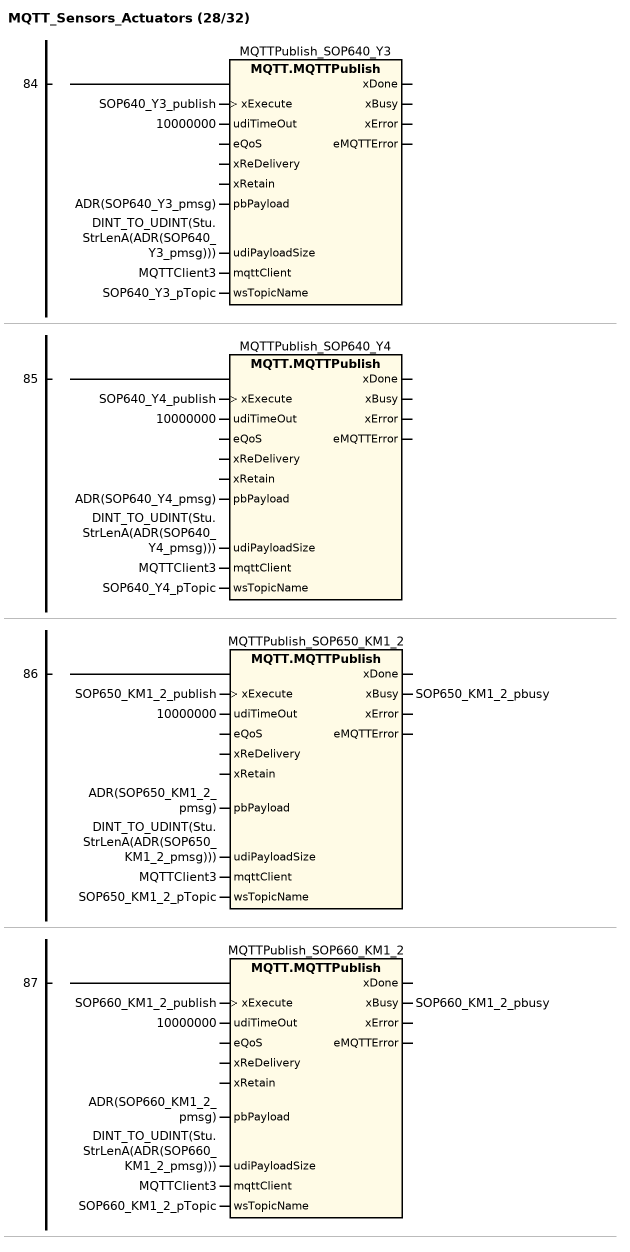
// NETWORK 84
_rt34(CLK := SOP640_Y3_publish);
MQTTPublish_SOP640_Y3(
    xExecute := _rt34.Q,
    udiTimeOut := 10000000,
    pbPayload := ADR(SOP640_Y3_pmsg),
    udiPayloadSize := DINT_TO_UDINT(Stu.StrLenA(ADR(SOP640_Y3_pmsg))),
    mqttClient := MQTTClient3,
    wsTopicName := SOP640_Y3_pTopic); // MQTT.MQTTPublish

// NETWORK 85
_rt35(CLK := SOP640_Y4_publish);
MQTTPublish_SOP640_Y4(
    xExecute := _rt35.Q,
    udiTimeOut := 10000000,
    pbPayload := ADR(SOP640_Y4_pmsg),
    udiPayloadSize := DINT_TO_UDINT(Stu.StrLenA(ADR(SOP640_Y4_pmsg))),
    mqttClient := MQTTClient3,
    wsTopicName := SOP640_Y4_pTopic); // MQTT.MQTTPublish

// NETWORK 86
_rt36(CLK := SOP650_KM1_2_publish);
MQTTPublish_SOP650_KM1_2(
    xExecute := _rt36.Q,
    udiTimeOut := 10000000,
    pbPayload := ADR(SOP650_KM1_2_pmsg),
    udiPayloadSize := DINT_TO_UDINT(Stu.StrLenA(ADR(SOP650_KM1_2_pmsg))),
    mqttClient := MQTTClient3,
    wsTopicName := SOP650_KM1_2_pTopic,
    xBusy => SOP650_KM1_2_pbusy); // MQTT.MQTTPublish

// NETWORK 87
_rt37(CLK := SOP660_KM1_2_publish);
MQTTPublish_SOP660_KM1_2(
    xExecute := _rt37.Q,
    udiTimeOut := 10000000,
    pbPayload := ADR(SOP660_KM1_2_pmsg),
    udiPayloadSize := DINT_TO_UDINT(Stu.StrLenA(ADR(SOP660_KM1_2_pmsg))),
    mqttClient := MQTTClient3,
    wsTopicName := SOP660_KM1_2_pTopic,
    xBusy => SOP660_KM1_2_pbusy); // MQTT.MQTTPublish

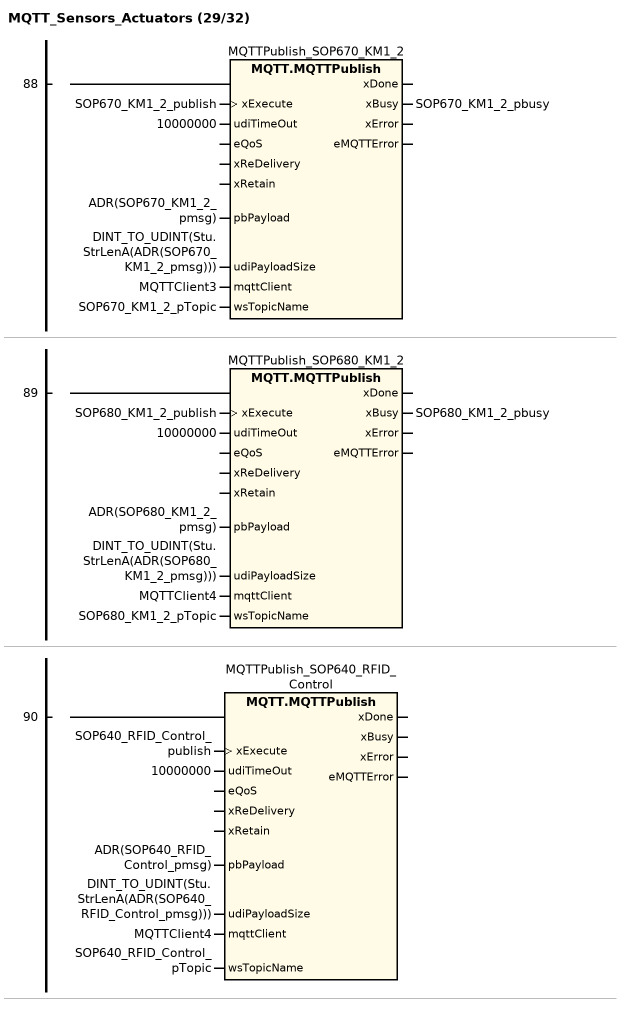
// NETWORK 88
_rt38(CLK := SOP670_KM1_2_publish);
MQTTPublish_SOP670_KM1_2(
    xExecute := _rt38.Q,
    udiTimeOut := 10000000,
    pbPayload := ADR(SOP670_KM1_2_pmsg),
    udiPayloadSize := DINT_TO_UDINT(Stu.StrLenA(ADR(SOP670_KM1_2_pmsg))),
    mqttClient := MQTTClient3,
    wsTopicName := SOP670_KM1_2_pTopic,
    xBusy => SOP670_KM1_2_pbusy); // MQTT.MQTTPublish

// NETWORK 89
_rt39(CLK := SOP680_KM1_2_publish);
MQTTPublish_SOP680_KM1_2(
    xExecute := _rt39.Q,
    udiTimeOut := 10000000,
    pbPayload := ADR(SOP680_KM1_2_pmsg),
    udiPayloadSize := DINT_TO_UDINT(Stu.StrLenA(ADR(SOP680_KM1_2_pmsg))),
    mqttClient := MQTTClient4,
    wsTopicName := SOP680_KM1_2_pTopic,
    xBusy => SOP680_KM1_2_pbusy); // MQTT.MQTTPublish

// NETWORK 90
_rt40(CLK := SOP640_RFID_Control_publish);
MQTTPublish_SOP640_RFID_Control(
    xExecute := _rt40.Q,
    udiTimeOut := 10000000,
    pbPayload := ADR(SOP640_RFID_Control_pmsg),
    udiPayloadSize := DINT_TO_UDINT(Stu.StrLenA(ADR(SOP640_RFID_Control_pmsg))),
    mqttClient := MQTTClient4,
    wsTopicName := SOP640_RFID_Control_pTopic); // MQTT.MQTTPublish

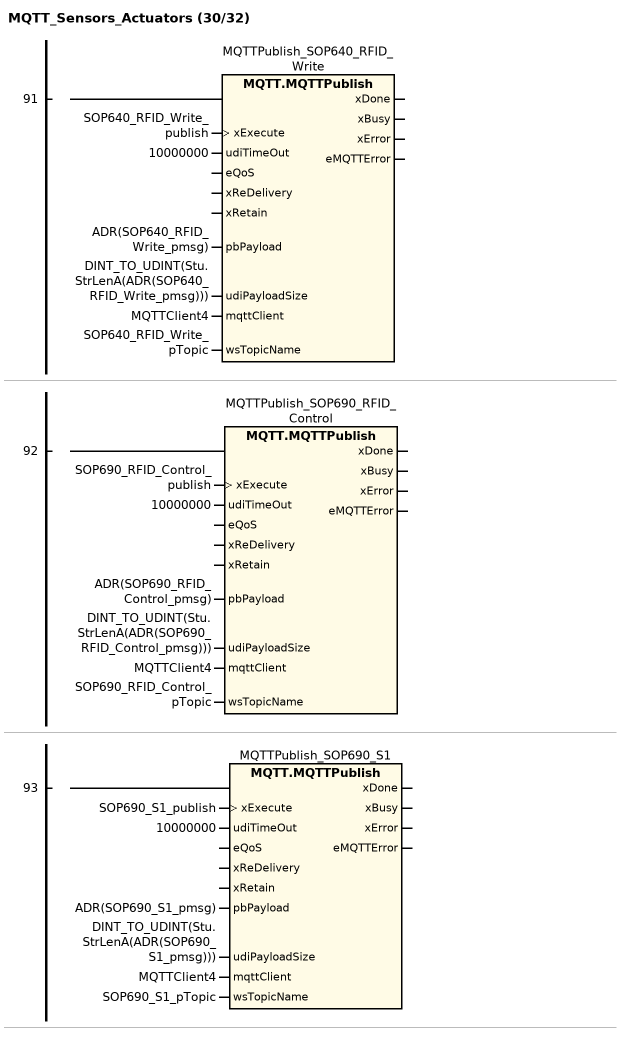
// NETWORK 91
_rt41(CLK := SOP640_RFID_Write_publish);
MQTTPublish_SOP640_RFID_Write(
    xExecute := _rt41.Q,
    udiTimeOut := 10000000,
    pbPayload := ADR(SOP640_RFID_Write_pmsg),
    udiPayloadSize := DINT_TO_UDINT(Stu.StrLenA(ADR(SOP640_RFID_Write_pmsg))),
    mqttClient := MQTTClient4,
    wsTopicName := SOP640_RFID_Write_pTopic); // MQTT.MQTTPublish

// NETWORK 92
_rt42(CLK := SOP690_RFID_Control_publish);
MQTTPublish_SOP690_RFID_Control(
    xExecute := _rt42.Q,
    udiTimeOut := 10000000,
    pbPayload := ADR(SOP690_RFID_Control_pmsg),
    udiPayloadSize := DINT_TO_UDINT(Stu.StrLenA(ADR(SOP690_RFID_Control_pmsg))),
    mqttClient := MQTTClient4,
    wsTopicName := SOP690_RFID_Control_pTopic); // MQTT.MQTTPublish

// NETWORK 93
_rt43(CLK := SOP690_S1_publish);
MQTTPublish_SOP690_S1(
    xExecute := _rt43.Q,
    udiTimeOut := 10000000,
    pbPayload := ADR(SOP690_S1_pmsg),
    udiPayloadSize := DINT_TO_UDINT(Stu.StrLenA(ADR(SOP690_S1_pmsg))),
    mqttClient := MQTTClient4,
    wsTopicName := SOP690_S1_pTopic); // MQTT.MQTTPublish

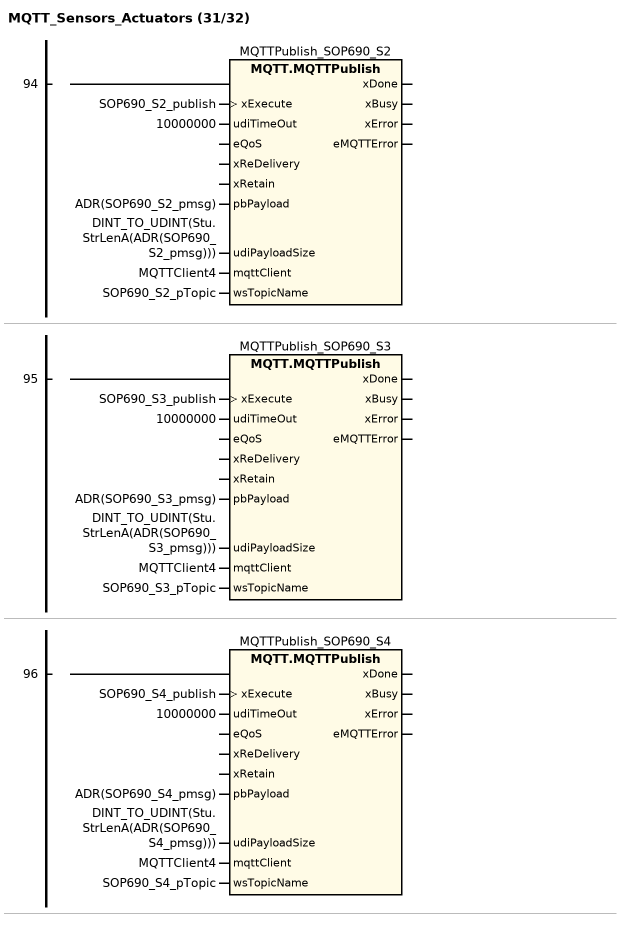
// NETWORK 94
_rt44(CLK := SOP690_S2_publish);
MQTTPublish_SOP690_S2(
    xExecute := _rt44.Q,
    udiTimeOut := 10000000,
    pbPayload := ADR(SOP690_S2_pmsg),
    udiPayloadSize := DINT_TO_UDINT(Stu.StrLenA(ADR(SOP690_S2_pmsg))),
    mqttClient := MQTTClient4,
    wsTopicName := SOP690_S2_pTopic); // MQTT.MQTTPublish

// NETWORK 95
_rt45(CLK := SOP690_S3_publish);
MQTTPublish_SOP690_S3(
    xExecute := _rt45.Q,
    udiTimeOut := 10000000,
    pbPayload := ADR(SOP690_S3_pmsg),
    udiPayloadSize := DINT_TO_UDINT(Stu.StrLenA(ADR(SOP690_S3_pmsg))),
    mqttClient := MQTTClient4,
    wsTopicName := SOP690_S3_pTopic); // MQTT.MQTTPublish

// NETWORK 96
_rt46(CLK := SOP690_S4_publish);
MQTTPublish_SOP690_S4(
    xExecute := _rt46.Q,
    udiTimeOut := 10000000,
    pbPayload := ADR(SOP690_S4_pmsg),
    udiPayloadSize := DINT_TO_UDINT(Stu.StrLenA(ADR(SOP690_S4_pmsg))),
    mqttClient := MQTTClient4,
    wsTopicName := SOP690_S4_pTopic); // MQTT.MQTTPublish

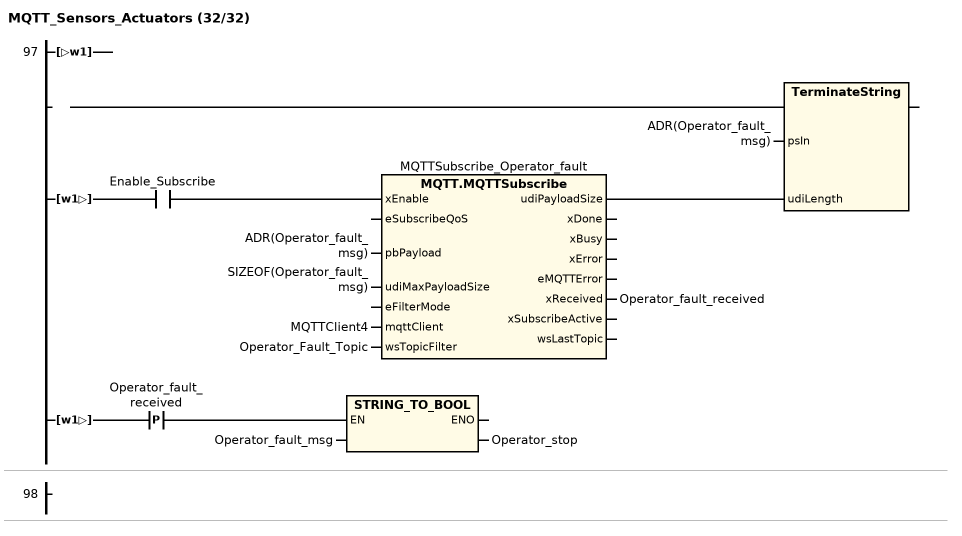
// NETWORK 97
MQTTSubscribe_Operator_fault(
    xEnable := Enable_Subscribe,
    pbPayload := ADR(Operator_fault_msg),
    udiMaxPayloadSize := SIZEOF(Operator_fault_msg),
    mqttClient := MQTTClient4,
    wsTopicFilter := Operator_Fault_Topic,
    xReceived => Operator_fault_received); // MQTT.MQTTSubscribe
TerminateString(psIn := ADR(Operator_fault_msg), udiLength := MQTTSubscribe_Operator_fault.udiPayloadSize);
_rt47(CLK := Operator_fault_received);
IF _rt47.Q THEN Operator_stop := STRING_TO_BOOL(Operator_fault_msg); END_IF

// NETWORK 98

END_PROGRAM

// Device/Application/FBs/TerminateString
// Terminates the STRING psIn at position udiLength
FUNCTION TerminateString : BOOL
VAR_INPUT
	psIn : POINTER TO BYTE; // Pointer to STRING
	udiLength : UDINT; // Length of psIn
END_VAR
VAR
END_VAR

psIn[udiLength] := 0;
TerminateString := TRUE;

END_FUNCTION

// Device/Application/Cases/Case1
PROGRAM Case1
VAR
	TON_0: TON;
	Equal: BOOL;
	Last_switch_msg: STRING(1024);
	Prueba: BOOL;
	R_TRIG_0: R_TRIG;
END_VAR
VAR // added by the converter: edge detectors and wires of the graphical bodies
    _rt1, _rt2 : R_TRIG;
    _w1, _w2, _w3, _w4 : BOOL;
    _ft1 : F_TRIG;
END_VAR

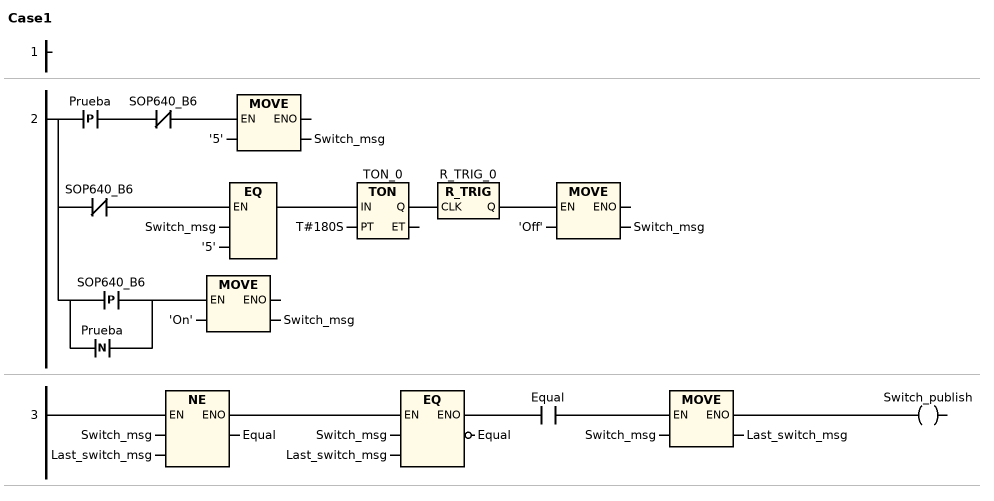
// NETWORK 1

// NETWORK 2
_rt1(CLK := Prueba);
_w1 := _rt1.Q AND NOT SOP640_B6;
IF _w1 THEN Switch_msg := '5'; END_IF
TON_0(IN := NOT SOP640_B6 AND Switch_msg = '5', PT := T#180S); // TON
R_TRIG_0(CLK := TON_0.Q); // R_TRIG
_w2 := R_TRIG_0.Q;
IF _w2 THEN Switch_msg := 'Off'; END_IF
_rt2(CLK := SOP640_B6);
_ft1(CLK := Prueba);
_w3 := _rt2.Q OR _ft1.Q;
IF _w3 THEN Switch_msg := 'On'; END_IF
(* _w1 OR _w2 OR _w3; result not used *)

// NETWORK 3
Equal := Switch_msg <> Last_switch_msg;
Equal := NOT (Switch_msg = Last_switch_msg);
_w4 := Equal;
IF _w4 THEN Last_switch_msg := Switch_msg; END_IF
Switch_publish := _w4;

END_PROGRAM

// Device/Application/Cases/Case2
PROGRAM Case2
VAR
	MQTTClient: MQTT.MQTTClient; 										// MQTTClient FB
	Port: UINT := 1883; 												// Port
	Will_msg: STRING(1024) := ''; 										// Message if there is disconnection
	Host: STRING(255) := '192.168.1.123'; 								// Broker IP 192.168.1.123 Simumatik
	Codesys: WSTRING(1024) := "codesys";								// Username and password "Codesys"
	Enable_Client: BOOL := TRUE; 										// Establishes connecting with the MQTT broker
	Enable_Subscribe: BOOL;												// Enables subscription
		
	MQTTPublish_SOP610_MC: MQTT.MQTTPublish;								// MQTTPublish FB
	SOP610_MC_publish: BOOL;
	SOP610_MC_pmsg: STRING(1024);
	SOP610_MC_pTopic: WSTRING(1024) := "OP60/SOP610_MC";	
	MQTTPublish_SOP620_MC: MQTT.MQTTPublish;								// MQTTPublish FB
	SOP620_MC_publish: BOOL;
	SOP620_MC_pmsg: STRING(1024);
	SOP620_MC_pTopic: WSTRING(1024) := "OP60/SOP620_MC";
	MQTTPublish_SOP630_MC: MQTT.MQTTPublish;								// MQTTPublish FB
	SOP630_MC_publish: BOOL;
	SOP630_MC_pmsg: STRING(1024);
	SOP630_MC_pTopic: WSTRING(1024) := "OP60/SOP630_MC";	
				 
	R_TRIG_0: R_TRIG;
	R_TRIG_1: R_TRIG;
	
	Publish1: BOOL;
	Publish2: BOOL;
	Prueba: BOOL;
END_VAR
VAR // added by the converter: edge detectors and wires of the graphical bodies
    _rt1, _rt2, _rt3 : R_TRIG;
    _w1, _w2, _w3 : BOOL;
    _ft1, _ft2 : F_TRIG;
END_VAR

